// TwinCAT 3 PLC project ExternControl
// ProgramVersion: 3.1.4026.26
// libraries:
//   Tc2_Standard, * (Beckhoff Automation GmbH)
//   Tc2_System, * (Beckhoff Automation GmbH)
//   Tc2_Utilities, * (Beckhoff Automation GmbH)
//   VisuDialogs, * (System)
//   VisuDialogs
// project tree:
//   APPLICATION/ MAIN_APP.TcPOU
//   / GlobalTextList.TcGTLO, MAIN.TcPOU (not stored), PlcTask.TcTTO (not stored), Visualization Manager.TcVMO (not stored)
//   MAPPING/ MAPPING_in.TcPOU (not stored), MAPPING_out.TcPOU (not stored)
//   MAPPING/_types/ U_APP_CTRL.TcDUT (not stored), U_APP_STATE.TcDUT (not stored), U_INSTANCE_CTRL.TcDUT (not stored), U_INSTANCE_STATE.TcDUT (not stored), U_TICKET_LIST_CTRL.TcDUT (not stored), U_TICKET_LIST_DATA_INPUT.TcDUT (not stored), U_TICKET_LIST_DATA_OUTPUT.TcDUT, U_TICKET_LIST_STATE.TcDUT (not stored), U_XTS_STATION_CTRL.TcDUT (not stored), U_XTS_STATION_STATE.TcDUT (not stored), U_XTS_TRANSPORT_CTRL.TcDUT (not stored), U_XTS_TRANSPORT_STATE.TcDUT (not stored)
//   PLC_MOTION/_GVL/ PLC_CONSTANT.TcGVL
//   XTS_TRANSPORT/CaGroup/types/ E_CA_GROUP_STATE.TcDUT, E_GROUP_CHECK.TcDUT, ST_GROUP_INFO.TcDUT
//   XTS_TRANSPORT/ GVL_XTS.TcGVL (not stored), GVL_XTS_CONSTANTS.TcGVL, GVL_XTS_VERSION.TcGVL (not stored)
//   XTS_TRANSPORT/Mover/types/ E_MOVER_CHECK.TcDUT, E_MOVER_CTRL.TcDUT, E_MOVER_SELECTOR.TcDUT, E_MOVER_STATE.TcDUT (not stored), ST_GEAR_DATA.TcDUT, ST_MOVER_CTRL.TcDUT, ST_MOVER_INFO.TcDUT (not stored), ST_MOVER_SELECTOR_CTRL.TcDUT, ST_MOVER_SELECTOR_STATE.TcDUT, ST_MOVER_STATE.TcDUT, ST_MOVE_DATA.TcDUT
//   XTS_TRANSPORT/Xpu/types/ E_XPU_CHECK.TcDUT, E_XPU_CTRL.TcDUT, E_XPU_INIT.TcDUT, E_XPU_STATE.TcDUT, ST_XPU_CTRL.TcDUT, ST_XPU_INFO.TcDUT, ST_XPU_STATE.TcDUT
//   XTS_TRANSPORT/XtsStation/types/ E_STATION_CHECK.TcDUT (not stored), E_STATION_CTRL.TcDUT, E_STATION_GEAR_DISTANCE_AXIS.TcDUT (not stored), E_STATION_STATE.TcDUT (not stored), E_STATION_TYPE.TcDUT (not stored), ST_STATION_CTRL.TcDUT (not stored), ST_STATION_GEAR_PARAMETER.TcDUT (not stored), ST_STATION_LIST_RESULT.TcDUT (not stored), ST_STATION_MOVER_DATA.TcDUT, ST_STATION_PARAMETER.TcDUT, ST_STATION_STATE.TcDUT (not stored), T_NEST_OFFSET.TcDUT (not stored)
//   XTS_TRANSPORT/XtsTransportUnit/types/ E_XTS_TRANSPORT_CHECK.TcDUT, E_XTS_TRANSPORT_CTRL.TcDUT, E_XTS_TRANSPORT_STATE.TcDUT, ST_XTS_TRANSPORT_CTRL.TcDUT, ST_XTS_TRANSPORT_STATE.TcDUT
//   XTS_TRANSPORT/_Visualization/ GROUP_VISU.TcVIS (not stored), MOVER_VISU.TcVIS (not stored), SELECTOR_VISU.TcVIS (not stored), STATION_VISU.TcVIS, XPU_VISU.TcVIS, XTS_TRANSPORT.TcVIS
//   XTS_TRANSPORT/_Visualization/textlists/ TL_E_CTRL_MOVER.TcTLO, TL_E_CTRL_STATION.TcTLO, TL_E_CTRL_TRANSPORT.TcTLO, TL_E_CTRL_XPU.TcTLO
//   XTS_TRANSPORT/_Visualization/types/ ST_XPU_STRINGS.TcDUT (not stored), T_MOVER_SELECTOR.TcVIS
//   _MSG/class/ fb_LocalTime.TcPOU, fb_MessageData.TcPOU, fb_MessageDataCtrl.TcPOU
//   _MSG/ f_MessageSet.TcPOU (not stored), GVL_MSG_AXIS.TcGVL (not stored), GVL_MSG_XTS.TcGVL, I_MessageData.TcIO
//   _MSG/types/ e_Device.TcDUT, E_MessageType.TcDUT, E_MESSAGE_BATCH.TcDUT, E_MESSAGE_CHECK.TcDUT, E_MESSAGE_CTRL.TcDUT (not stored), E_MESSAGE_FLOW.TcDUT, E_MESSAGE_STATE.TcDUT, e_Subdevice.TcDUT, ST_Message.TcDUT, ST_MESSAGE_CTRL.TcDUT (not stored), ST_MESSAGE_STATE.TcDUT (not stored), TL_E_MESSAGETYPE.TcTLO
//   _types/ E_CHECK_STATE.TcDUT, E_PROGRESS.TcDUT, f_GetProgress.TcPOU (not stored), f_GetState.TcPOU
// (motion and I/O tree: see PLC project xtstransport)
// real-time tasks:
//   TASK XTS Task 1: cycle T#250us, priority 1, ADS port 350
//   TASK PLC_1: cycle T#2ms, priority 15, ADS port 353
//   TASK Job Task: cycle default, priority 32
// variable links:
//   ExternControl/ExternControl Instance <-> XtsTransport/XtsTransport Instance
//     PlcTask Inputs/MAIN_APP.eInitXts <-> PlcTask Outputs/MAIN_APP.eInit
//     PlcTask Inputs/MAPPING_in.StationState.byState <-> PlcTask Outputs/MAPPING_XTS_out.StationState.byState
//     PlcTask Inputs/MAPPING_in.TransportState.byState <-> PlcTask Outputs/MAPPING_XTS_out.TransportState.byState
//     PlcTask Outputs/MAPPING_out.StationControl.byCtrl <-> PlcTask Inputs/MAPPING_XTS_in.StationControl.byCtrl
//     PlcTask Outputs/MAPPING_out.TransportControl.byCtrl <-> PlcTask Inputs/MAPPING_XTS_in.TransportControl.byCtrl

// ---- MAPPING/_types/U_TICKET_LIST_DATA_OUTPUT.TcDUT
TYPE U_TICKET_LIST_DATA_OUTPUT :
UNION
  stData              : ST_LIST_NODE_DATA;
  byData   AT %I*     : ARRAY[1..SIZEOF(ST_LIST_NODE_DATA)] OF BYTE;
END_UNION
END_TYPE

// ---- XTS_TRANSPORT/CaGroup/types/E_CA_GROUP_STATE.TcDUT
// {attribute 'qualified_only'}
// {attribute 'strict'}
{attribute 'to_string'}
TYPE E_CA_GROUP_STATE :
(
  // replicated from MC_GROUP_STATE for getting to_string() functionality
	mcGroupStateInvalid   :=0, 
  mcGroupStateDisabled  :=1, 
  mcGroupStateStandby   :=2, 
  mcGroupStateMoving    :=3, 
  mcGroupStateStopping  :=4, 
  mcGroupStateErrorStop :=5, 
  mcGroupStateHoming    :=6, 
  mcGroupStateNotReady  :=7, 
  mcGroupStateSuspended :=8 
)UINT;
END_TYPE

// ---- XTS_TRANSPORT/CaGroup/types/E_GROUP_CHECK.TcDUT
{attribute 'qualified_only'}
{attribute 'to_string'}
TYPE E_GROUP_CHECK :
(
  NULL,
  REFERENCE_GROUP_REF_INVALID := 9000,
  REFERENCE_AXIS_REF_INVALID,
  REFERENCE_CTRL_INVALID,
  REFERENCE_STATE_INVALID,
  REFERENCE_MOVER_ITF_INVALID,
  REFERENCE_XPU_INFO_INVALID,

  CHECK_DONE              := 10000
)UINT;
END_TYPE

// ---- XTS_TRANSPORT/CaGroup/types/ST_GROUP_INFO.TcDUT
TYPE ST_GROUP_INFO :
STRUCT
  GroupStatusValid,
  GroupStatusBusy,
  GroupMoving, 
  GroupHoming, 
  GroupErrorStop, 
  GroupNotReady, 
  GroupStandby, 
  GroupStopping,
 
  GroupDisabled, 
  AllAxesStanding, 
  ConstantVelocity, 
  Accelerating, 
  Decelerating, 
  InPosition, 
  GroupError					  : BIT; 

  GroupErrorId					: UDINT;

  AxisCount      				: UDINT;
  AxisCountEnabled      : UDINT;

  {attribute 'displaymode':='hex'}
  CaGroupOID            : OTCID;

  CaGroupState          : E_CA_GROUP_STATE;
END_STRUCT
END_TYPE

// ---- XTS_TRANSPORT/Mover/types/E_MOVER_CHECK.TcDUT
{attribute 'qualified_only'}
{attribute 'strict'}
{attribute 'to_string'}
TYPE E_MOVER_CHECK :
(
  NULL,
  MOVER_ID_INVALID := 9000,
  REFERENCE_AXIS_REF_INVALID,
  REFERENCE_LAST_POSITION_INVALID,
  REFERENCE_LAST_GAP_INVALID,
  REFERENCE_INFO_INVALID,

  REFERENCE_CTRL_INVALID  := 9100,
  REFERENCE_STATE_INVALID,
  REFERENCE_GEAR_DATA_INVALID,
  REFERENCE_MOVE_DATA_INVALID,
  REFERENCE_MOVER_ITF_INVALID,

  CHECK_DONE  := 10_000
)UINT;
END_TYPE

// ---- XTS_TRANSPORT/Mover/types/E_MOVER_CTRL.TcDUT
{attribute 'qualified_only'}
{attribute 'strict'}
{attribute 'to_string'}
TYPE E_MOVER_CTRL :
(
  MOVER_NULL,               // initial value at startup, used for change of order or retrigger
  MOVER_ENABLE,             // sets MC_Power.Enable
  MOVER_DISABLE,            // removes MC_Power.Enable
  MOVER_MOVE_TO_POS,        // modulo absolute positioning with MC_MoveAbsolute, InTargetPosition check
  MOVER_MOVE_TO_POS_CA,     // modulo absolute positioning with MC_MoveAbsoluteCA, InTargetPosition check
  MOVER_SEND_TO_POS_CA,     // modulo absolute positioning with MC_MoveAbsoluteCA, done after moving ReleaseDistance
  MOVER_HALT,               // halts mover; by use of MC_Halt mover is set passive in CA group
  MOVER_GEAR_IN,            // GearIn for mover in standstill

  MOVER_GEAR_IN_POS_CA,     // GearInPosCA of mover; when FB_GearInPosCa is InSync --> order is done; check SyncDistance yourself and release mover with e_mover_order.mover_SendToPos
  MOVER_GEAR_OUT,           // gear out for mover
  MOVER_RESET,              // MC_RESET for mover
  MOVER_INFO                // used to display MoverInfo in ST_MOVER_SELECTOR_STATE.Info
)UINT;
END_TYPE

// ---- XTS_TRANSPORT/Mover/types/E_MOVER_SELECTOR.TcDUT
{attribute 'qualified_only'}
{attribute 'strict'}
{attribute 'to_string'}
TYPE E_MOVER_SELECTOR :
(
	SELECT_MOVER_INDEX,
  SELECT_MOVER_AXIS_ID
);
END_TYPE

// ---- XTS_TRANSPORT/Mover/types/ST_GEAR_DATA.TcDUT
{attribute 'pack_mode' := '2'}
TYPE ST_GEAR_DATA :
STRUCT
  rDeltaToMasterPos       : LREAL;
  rModuloSyncPosSlave     : LREAL;
  rMasterStartDistance    : LREAL;
  rGearNumerator          : LREAL;
  iGearDenumerator        : USINT  := 1;
END_STRUCT
END_TYPE

// ---- XTS_TRANSPORT/Mover/types/ST_MOVER_CTRL.TcDUT
{attribute 'pack_mode' := '2'}
TYPE ST_MOVER_CTRL :
STRUCT
  Cmd             : E_MOVER_CTRL;  // order to execute on mover
END_STRUCT
END_TYPE

// ---- XTS_TRANSPORT/Mover/types/ST_MOVER_SELECTOR_CTRL.TcDUT
TYPE ST_MOVER_SELECTOR_CTRL :
STRUCT
  Selector      : E_MOVER_SELECTOR; // select by array Index OR AXIS_REF.NcToPlc.AxisId 
  Mover         : UINT;             // array Index OR AXIS_REF.NcToPlc.AxisId
  Control       : ST_MOVER_CTRL;    // mover control struct, put motion command in here

  Data          : ST_MOVE_DATA;     // write your movement parameters
  //Gear          : ST_GEAR_DATA;     // write your gearing parameters
END_STRUCT
END_TYPE

// ---- XTS_TRANSPORT/Mover/types/ST_MOVER_SELECTOR_STATE.TcDUT
TYPE ST_MOVER_SELECTOR_STATE :
STRUCT
  MoverIndex  : UINT;
  AxisId      : UDINT;
  State       : ST_MOVER_STATE;

  Info        : ST_MOVER_INFO;
END_STRUCT
END_TYPE

// ---- XTS_TRANSPORT/Mover/types/ST_MOVER_STATE.TcDUT
{attribute 'pack_mode' := '2'}
TYPE ST_MOVER_STATE :
STRUCT
  State           : E_MOVER_STATE;  // ST_MOVER_CTRL.Cmd with added E_PROGRESS
  MasterId        : USINT;            // mirror NC AxisId of Master axis
END_STRUCT
END_TYPE

// ---- XTS_TRANSPORT/Mover/types/ST_MOVE_DATA.TcDUT
{attribute 'pack_mode' := '2'}
TYPE ST_MOVE_DATA :
STRUCT
  // HAUD 2024 03 14
  // some init data added for example
  rPos            : LREAL :=   2275.0;
  rVelo           : LREAL :=    500.0;
  rAcc            : LREAL :=   5000.0;
  rJerk           : LREAL := 500000.0;
  rGap            : LREAL :=    100.0;
  rOverride       : LREAL :=    100.0;
  rDelta          : LREAL :=      0.05;
  rDistance       : LREAL :=     25.0;
END_STRUCT
END_TYPE

// ---- XTS_TRANSPORT/Xpu/types/E_XPU_CHECK.TcDUT
{attribute 'qualified_only'}
{attribute 'to_string'}
TYPE E_XPU_CHECK :
(
  INIT_CHECK,
  INIT_CHECK_ERROR,
  START_CHECK,
  XPU_INSTANCE_NULL,
  XPU_RAIL_LENGTH,
  GROUP_RAIL_LENGTH,
  RAIL_LENGTH_COMPARE,
  GROUP_NOT_CONFIGURED,
  GROUP_OID_MISMATCH,

  MOVER_COUNT             := 10,
  MOVER_COUNT_ZERO,
  MOVER_COUNT_NOT_EQUAL,

  PROCESSING_UNIT_POSITIONS_VALID         := 20,
  PROCESSING_UNIT_GET_DATA_EXCEED,

  MOVER_ID_STANDARD       := 30,
  MOVER_ID_SIMULATION,
  MOVER_ID_DETECTION_MODE,
  MOVER_ID_DETECTION_VALID,
  MOVER_ID_DETECTION_DC_LINK,
  MOVER_ID_DETECTION_BUSY,
  MOVER_ID_DETECTION_IDLE,
  MOVER_ID_DETECTION_STATE,
  MOVER_ID_MULTIPLE_NOT_SUPPORTED,

  POINTER_CHECK           := 90,
  POINTER_NULL_CTRL,
  POINTER_NULL_STATE,

  CHECK_DONE      := 10_000
)UINT;
END_TYPE

// ---- XTS_TRANSPORT/Xpu/types/E_XPU_CTRL.TcDUT
{attribute 'strict'}
TYPE E_XPU_CTRL :
(
  XTS_CMD_NULL,
  XTS_CMD_INIT                  := 10,
  //XTS_CMD_READ_STN_CONFIG       := 20,
  XTS_IDLE                      := 30
)UINT;
END_TYPE

// ---- XTS_TRANSPORT/Xpu/types/E_XPU_INIT.TcDUT
{attribute 'to_string'}
TYPE E_XPU_INIT :
(
	INIT_START,
  INIT_ENVIRONMENT_OID            := 10,
  INIT_INFO_SERVER_ITF,
  INIT_INFO_SERVER_STATION_COUNT,
  INIT_INFO_SERVER_STATION_OID,
  INIT_CA_GROUP_OID               := 20,
  INIT_CA_GROUP_GET_OID,
  INIT_CA_GROUP_CHECK_OID,
  INIT_CA_GROUP_COM,
  INIT_PARAMETERSET_COUNT,
  INIT_PARAMETERSET_OID,
  INIT_PARAMETERSET_COM,
  INIT_PARAMETERSET_COM_INIT,
  INIT_PARAMETERSET_COM_NEXT,
  INIT_PROCESSING_UNIT_COM        := 30,
  INIT_PROCESSING_UNIT_COM_INIT,
  INIT_PROCESSING_UNIT_PART_COUNT,
  INIT_PROCESSING_UNIT_PART_OID,
  INIT_PROCESSING_UNIT_TRACK_COUNT,
  INIT_PROCESSING_UNIT_TRACK_OID,
  INIT_PROCESSING_UNIT_MOVER_COUNT,
  INIT_PROCESSING_UNIT_MOVER_OID,
  INIT_PROCESSING_UNIT_TASK_COUNT,
  INIT_PROCESSING_UNIT_TASK_OID,
  INIT_TRACK_COM                  := 50,
  INIT_TRACK_COM_INIT,
  INIT_PART_COM                   := 60,
  INIT_PART_COM_INIT,
  INIT_PART_MODULE_COUNT,
  INIT_PART_MODULE_OID,
  INIT_PART_MODULE_COM,
  INIT_PART_MODULE_COM_INIT,
  INIT_PART_MODULE_COM_NEXT,
  INIT_MOVER_COM                  := 70,
  INIT_MOVER_COM_INIT,
  INIT_MOVER_COM_NEXT,
  INIT_NCT_CONTROLLER_OID         := 80,
  INIT_NCT_CONTROLLER_COM,
  INIT_NCT_CONTROLLER_COM_INIT,
  INIT_NCT_BASE_UNIT_COUNT,
  INIT_NCT_BASE_UNIT_ITF,
  INIT_NCT_BASE_UNIT_NEXT,
  INIT_DATA_GET                   := 90,
  INIT_DATA_CHECK,
  INIT_DONE                       := 100
)UINT;
END_TYPE

// ---- XTS_TRANSPORT/Xpu/types/E_XPU_STATE.TcDUT
{attribute 'to_string'}
TYPE E_XPU_STATE :
(
  XTS_NULL,
  XTS_INVALID,
  XTS_INIT                      := 10,    // initialize XPU
  XTS_STATION_INFO_READ         := 20,    // get Station information from Xpu
  XTS_IDLE                      := 30
)UINT;
END_TYPE

// ---- XTS_TRANSPORT/Xpu/types/ST_XPU_CTRL.TcDUT
{attribute 'pack_mode' := '2'}
TYPE ST_XPU_CTRL :
STRUCT
  Cmd             : E_XPU_CTRL;
END_STRUCT
END_TYPE

// ---- XTS_TRANSPORT/Xpu/types/ST_XPU_INFO.TcDUT
{attribute 'pack_mode' := '2'}
TYPE ST_XPU_INFO :
STRUCT
  AllPositionsValid   : BIT;
  IdDetectionError    : BIT;
  IdDetectionValid    : BIT;
  IdDetectionActive   : BIT;

  OperationMode       : UINT;

  IdDetectionMode           : UINT;
  MoverPositionAssignement  : UINT;

  nDetectedAxisCount  : UINT;
  nExpectedAxisCount  : UINT;

  nParameterSetCount  : UINT;
  nModuleCount        : UINT;
  rRailLength         : LREAL;
END_STRUCT
END_TYPE

// ---- XTS_TRANSPORT/Xpu/types/ST_XPU_STATE.TcDUT
{attribute 'pack_mode' := '2'}
TYPE ST_XPU_STATE :
STRUCT
  Init            : E_XPU_INIT;
  State           : E_XPU_STATE;
  Check           : E_XPU_CHECK;  // cyclic check result
  DcLink          : BIT;          // power all motor modules is ON
END_STRUCT
END_TYPE

// ---- XTS_TRANSPORT/XtsStation/types/E_STATION_CTRL.TcDUT
{attribute 'qualified_only'}
{attribute 'strict'}
{attribute 'to_string'}
TYPE E_STATION_CTRL :
(
  STATION_CTRL_NULL,              // nothing happens here
	STATION_INIT            := 1,   // hard reset of station, list is cleared
  STATION_DISABLE         := 10,  // 
  STATION_ENABLE,                 // 

  STATION_MOVER_ENTER     := 20,  // mover may enter station
  STATION_MOVER_ENTER_RETRY,      // retry after E_STATION_STATE.STATION_ERROR_INFEED_ERROR
  STATION_MOVER_SEND,             // do not enter, send to E_STATION_STATE.STATION_MOVER_OUT

  STATION_PROCESS_START   := 30,  // double handshake with extern
  STATION_PROCESS_DONE,           // single handshake with extern
  STATION_PROCESS_NEST_SKIP,

  STATION_MOVER_OUT       := 50,  // mover may leave station now; ticket for mover is checked here (ST_STATION_CTRL.nTargetStation)
  STATION_MOVER_OUT_RETRY,        // retry after E_STATION_STATE.STATION_ERROR_OUTFEED_ERROR

  STATION_MOVER_GONE      := 60   // mover has left station, last handshake station is empty

)USINT;
END_TYPE

// ---- XTS_TRANSPORT/XtsStation/types/ST_STATION_MOVER_DATA.TcDUT
{attribute 'pack_mode' := '2'}
TYPE ST_STATION_MOVER_DATA :
STRUCT
  nMoverId        : USINT;  // who am I?  !! MUST be correct !! - movement to base position sets everything in order, DO NOT manipulate!
  nTargetStation  : USINT;  // where shall I be? used for double checking with StationId at infeed of mover into station

  {attribute 'displaymode':='bin'}
  nMask           : BYTE;   // how many of you are there? (1 = default, no action required)

  rOffset         : REAL;   // offset for use in work flow !! added to static mover offset for every nest(bit) in nMask!!
END_STRUCT
END_TYPE

// ---- XTS_TRANSPORT/XtsStation/types/ST_STATION_PARAMETER.TcDUT
TYPE ST_STATION_PARAMETER :
STRUCT
  eType             : E_STATION_TYPE := 1;  // StationProcess or StationGearInPos
  sText             : STRING(80);           // only description
  rPosWait          : REAL;                 // start of station, 
                                            // a sending station is using this value 
                                            // to send mover to

  rReleaseDistance  : REAL;                 // distance mover has to travel (from ActPos) 
                                            // in order for station to go back to disable

  rGap              : REAL;
  rVelo             : REAL;
  rAccDec           : REAL;
  rJerk             : REAL;

  // how many nests (stop positions) mover has to stop at (1 = default)
  nConfiguredStopCount  : USINT := 1; // 1-8 --> NestMask = BYTE

  // mover stop position in station, relative to rPosWait!!
  rPosStop          : ARRAY[1..8] OF LREAL;
END_STRUCT
END_TYPE

// ---- XTS_TRANSPORT/XtsTransportUnit/types/E_XTS_TRANSPORT_CHECK.TcDUT
{attribute 'qualified_only'}
{attribute 'to_string'}
TYPE E_XTS_TRANSPORT_CHECK :
(
  // info for cyclic checks
  INIT_CHECK,
  START_CHECK,    // check cycle start
  XPU_INIT,       // Xpu: initialization


  // errors in fb_TransportUnit.Check()
  POINTER_CHECK           := 9000,
  POINTER_NULL_CTRL,

  POINTER_NULL_STATE,
  POINTER_NULL_XPU_CTRL,

  POINTER_NULL_XPU_STATE,
  POINTER_NULL_XPU_INFO,

  POINTER_NULL_GROUP_ITF,
  POINTER_NULL_GROUP_INFO,

  POINTER_NULL_MOVER,
  POINTER_NULL_MOVER_ITF,

  POINTER_NULL_MOVER_INFO,
  POINTER_NULL_MOVER_LAST_POS,
  POINTER_NULL_MOVER_LAST_GAP,

  POINTER_NULL_STATION_START,
  POINTER_NULL_STATION_ITF,
  POINTER_NULL_STATION_CONTROL,
  POINTER_NULL_STATION_STATE,
  POINTER_NULL_STATION_CTRL_ITF,

  DONE_CHECK              := 10000
)UINT;
END_TYPE

// ---- XTS_TRANSPORT/XtsTransportUnit/types/E_XTS_TRANSPORT_CTRL.TcDUT
{attribute 'strict'}
{attribute 'to_string'}
TYPE E_XTS_TRANSPORT_CTRL :
(
  CMD_NULL,
  CMD_INIT                  := 10,  // Xpu, Group, Mover initialization: clear errors, clear group, check Xpu data, check mover detection
  CMD_IDLE,

  CMD_MOVER_ENABLE          := 20,  // all mover are enabled, checked for ControlLoopClosed
  CMD_MOVER_DISABLE,                // all mover are disabled, no axis in CaGroup: no error, any axis in CaGroup: group error
  CMD_MOVER_HALT_CA,                // all movers are stopped with MC_HaltCA[]. ONLY use if all movers are in CA group
  CMD_MOVER_STOP,

  CMD_GROUP_CLEAR           := 30,  // halt all movers, clear errors, remove all movers from group, clear group
  CMD_GROUP_BUILD,                  // add all movers to group
  CMD_GROUP_ENABLE,                 // group with movers is enabled
  CMD_GROUP_STOP,                   // moving CA Group is stopped

  CMD_TRANSPORT_START       := 40,  // move all mover[i] to start position
  CMD_TRANSPORT_RESTART             // move all mover[i] to LastPosition[i]

)UINT;
END_TYPE

// ---- XTS_TRANSPORT/XtsTransportUnit/types/E_XTS_TRANSPORT_STATE.TcDUT
{attribute 'to_string'}
TYPE E_XTS_TRANSPORT_STATE :
(
  TRANSPORT_NULL,
  TRANSPORT_INVALID,
  TRANSPORT_INIT            := 10,  // Xpu, Group, Mover initialization: init TcCOM objects, clear errors, clear group, check Xpu data, check mover detection
  TRANSPORT_IDLE,                   // cyclic check for errors, check Xpu data

  TRANSPORT_MOVER_ENABLE    := 20,  // all mover are enabled, checked for ControlLoopClosed
  TRANSPORT_MOVER_DISABLE,          // all mover are disabled
  TRANSPORT_MOVER_HALT_CA,          // all mover standstill
  TRANSPORT_MOVER_STOP,

  TRANSPORT_GROUP_CLEAR     := 30,  // halt all movers, clear errors, remove all movers from group, clear group
  TRANSPORT_GROUP_BUILD,            // add all movers to group
  TRANSPORT_GROUP_ENABLE,           // group with movers is enabled
  TRANSPORT_GROUP_STOP,             // CaGroup Stop, CaGroup Reset, All movers halt

  TRANSPORT_START           := 40,  // move all mover[i] to start position
  TRANSPORT_RESTART                 // move all mover[i] to LastPosition[i]
)UINT;
END_TYPE

// ---- XTS_TRANSPORT/XtsTransportUnit/types/ST_XTS_TRANSPORT_CTRL.TcDUT
{attribute 'pack_mode' := '2'}
TYPE ST_XTS_TRANSPORT_CTRL :
STRUCT
  Cmd       : E_XTS_TRANSPORT_CTRL;
END_STRUCT
END_TYPE

// ---- XTS_TRANSPORT/XtsTransportUnit/types/ST_XTS_TRANSPORT_STATE.TcDUT
{attribute 'pack_mode' := '2'}
TYPE ST_XTS_TRANSPORT_STATE :
STRUCT
  State         : E_XTS_TRANSPORT_STATE;  // combined value of state and result(e_progress); (hint: extract state value by mod division)
  Check         : E_XTS_TRANSPORT_CHECK;

  XpuState      : ST_XPU_STATE;
  XpuInfo       : ST_XPU_INFO;
  GroupInfo     : ST_GROUP_INFO; 
END_STRUCT
END_TYPE

// ---- _MSG/types/e_Device.TcDUT
{attribute 'to_string'}
TYPE e_Device :
(
  Device_Null,                  // NULL               - not to be used
  Device_Main,                  // MAIN(PRG)          - reserved for MAIN(PRG)
  Device_MainAxis,              // MAIN_AXIS(PRG)     - reserved for MAIN_AXIS(PRG)
  Device_Nci,                   // NCI(PRG)           - reserved for NCI(PRG)
  Device_Cam,                   // CAM(PRG            - reserved for CAM(PRG)
  Device_Functions,             // FUNCTIONS(PRG)     - reserved for FUNCTIONS(PRG)
  Device_FlyingSaw,             // FLYING_SAW(PRG)    - reserved for FLYING_SAW(PRG)
  Device_MainApplication,       // MAIN_APP(PRG)      - reserved for MAIN_APP(PRG)

  Device_MoverSelector,         // single mover interface for xts applications
  Device_ParameterSelector,     // fb_ParameterSelector can only exist once in a project.
  Device_Configuration,         // fb_Configuration can handle multiple files therefore only one instance is required
  Device_XmlData,               // generic XML Data (e.g. persistent data)
  Device_Utilities,             // service calls to anyone you may want to talk to, the main intent is to get XPU and TcXtsIo data to the application side

  General           :=  1000,
  CaGroup           :=  2000,
  Xpu               :=  3000,
  XpuCtrl           :=  4000,
  Mover             :=  5000,
  MoverCtrl         :=  6000,
  XtsTransportUnit  :=  7000,
  XfcTriggerBox     :=  8000,
  XfcTouchProbe     :=  9000,
  XtsStation        := 10000,

  Camming           := 11000,
  NciChannel        := 12000,
  NciChannelCtrl    := 13000,
  Axis              := 14000,
  XfcAxis           := 15000,

  // txt file logging LOG_FILE_METRICS
  MetricsXts        := 16000,   //entries from xts Metrics are written into dedicated txt file (see f_MessageSet, here's the diverter)
  MetricsAxis       := 17000,   //entries from PLC_MOTION Metrics are written into dedicated txt file

  // txt file logging LOG_FILE_APP
  Process           := 20000,   // entries from process are written into dedicated txt file.
  ProcessListCtrl   := 21000,
  TicketListCtrl    := 22000,

  Application       := 30000,   // entries from application are written into dedicated txt file.


  // txt file logging LOG_FILE_PRODUCT - this is for you to use
  DataProduct       := 40000
)UDINT;
END_TYPE

// ---- _MSG/types/E_MessageType.TcDUT
{attribute 'strict'}
{attribute 'to_string'}
TYPE E_MessageType :
(
  //-----------------------------------------------------
  //-----------------------------------------------------
  //  message system:
  //  - errors are always calling f_MessageSet()
  //  - errors are always entered into its list
  //
  //  - message severity is set by this enum (like everywhere else)
  //
  //  - message frequency is set by this enum
  //    - IF you get above 50 stations, 
  //      writing to the file system takes time:
  //
  //    Batch: switching on metrics (> Empty) must not add cpu load, 
  //      --> so do not clutter here
  //
  //    Info:  regular flow of information (>Error / >Warning) 
  //           must not add significant cpu load, 
  //      --> so do not clutter here
  //
  //    Verbose and above:
  //    --> for small systems (< 96 mover, < 50 stations) 
  //        you may switch it on for everybody, 
  //        files get big quickly ;-)
  //
  //    --> switch on during test phase for a handful of stations
  //
  //    --> high detail logging always and for everybody
  //    --> we need somebody who transfers data more quickly
  //      --> I can offer a .NET(C#) ADS tool which collects the list.
  //          .NET application then pushes to database
  //-----------------------------------------------------
  //-----------------------------------------------------
  eMessageEmpty,    // he who is without bounds may speak
  eMessageBatch,    // he who counts words, counts numbers (Batch started, Next in Batch, Batch done)
  eMessageError,    // mine, your(')s, anybody's, let the numbers tell you
  eMessageWarning,  // I told you so
  eMessageInfo,     // A long time ago in a galaxy far, far away...
  eMessageVerbose,  // He talks a lot, doesn't he?; Yeah! He's very knowledgeable.
  eMessageSentient  // Keep them out of bright light, Don't get them wet, do not feed them after midnight!! No matter how much they beg!!
)DINT;
END_TYPE

// ---- _MSG/types/E_MESSAGE_BATCH.TcDUT
{attribute 'qualified_only'}
{attribute 'strict'}
{attribute 'to_string'}
TYPE E_MESSAGE_BATCH :
(
	MSG_BATCH_NULL,
  MSG_BATCH_JOB_STARTED,
  MSG_BATCH_NEXT_IN_JOB,
  MSG_BATCH_JOB_DONE
)UINT;
END_TYPE

// ---- _MSG/types/E_MESSAGE_CHECK.TcDUT
{attribute 'qualified_only'}
{attribute 'strict'}
{attribute 'to_string'}
TYPE E_MESSAGE_CHECK :
(
  NULL,
  // 9000 --> here comes your error
  POINTER_INVALID             := 9000,
  POINTER_TIME_INVALID,
  POINTER_LIST_INVALID,
  POINTER_MSG_IDX_INVALID,
  POINTER_ERR_IDX_INVALID,
  POINTER_ROOT_FILE_INVALID,
  POINTER_ROOT_DIR_INVALID,
  POINTER_CTRL_INVALID,
  POINTER_STATE_INVALID,

  // 10000 --> here comes your man
  CHECK_DONE                        := 10000
)UINT;
END_TYPE

// ---- _MSG/types/E_MESSAGE_FLOW.TcDUT
{attribute 'qualified_only'}
{attribute 'strict'}
{attribute 'to_string'}
TYPE E_MESSAGE_FLOW :
(
  MSG_FLOW_INIT,
  MSG_FLOW_ROOT                 := 10,
  MSG_FLOW_ROOT_CREATE,
  MSG_FLOW_ROOT_CREATE_BUSY,
  MSG_FLOW_FOLDER,
  MSG_FLOW_FOLDER_CREATE,
  MSG_FLOW_FOLDER_CREATE_BUSY,
  MSG_FLOW_FILE_CREATE_DONE,
  MSG_FLOW_LINE_START           := 100,
  MSG_FLOW_LINE_BUILD,
  MSG_FLOW_LINE_CHECK,
  MSG_FLOW_WRITE_FILE_BUSY      := 200,
  MSG_FLOW_WRITE_FILE_END,
  MSG_FLOW_WRITE_FILE_DONE      := 1000
)UINT;
END_TYPE

// ---- _MSG/types/E_MESSAGE_STATE.TcDUT
{attribute 'qualified_only'}
//{attribute 'strict'}
{attribute 'to_string'}
TYPE E_MESSAGE_STATE :
(
	MSG_STATE_NULL,
  MSG_STATE_INIT    := 10,
  MSG_STATE_IDLE    := 30,
  MSG_STATE_WRITE   := 50
)UINT;
END_TYPE

// ---- _MSG/types/e_Subdevice.TcDUT
{attribute 'strict'}
{attribute 'to_string'}
TYPE e_Subdevice :
(
  // sub device for message system
  General                 :=  0,
  MainInit,
  // Motion Control FB Instances
  fbPower,
  fbReset,
  fbResetSercos,
  fbHalt,
  fbStop,                 // 5
  fbHome,
  fbJog,
  fbMoveVelocity1,
  fbMoveVelocity2,
  fbMoveAbsolute1,        // 10
  fbMoveAbsolute2,
  fbMoveEndless,
  fbMovePtP,
  fbMoveVelo,
  fbSendToPos,

  // CA CollisionAvoidance FB instances
  // CA group fb instances
  fbCaGroup             := 30,
  fbMoveToPosCa,
  fbSendToAbsPosCa,
  fbSendToModuloPosCa,
  fbGearInPosCa,
  fbGroupAddAxis,
  fbGroupRemoveAxis,
  fbGroupDisable,
  fbGroupEnable,
  fbGroupErrorRead,
  fbGroupStatusRead,
  fbGroupReset,
  fbGroupStop,
  fbHaltCa,

  fbGearIn                := 50,
  fbGearOut,
  fbGearInMultiMaster,

  fbCamOutV2              := 80,
  fbCamInV2,
  fbCamScalingV2,
  fbCamInfoV2,
  fbReadMotionFunction,
  fbReadMotionFunctionPoint,
  fbReadMotionFunctionValues,
  fbWriteMotionFunction,
  fbWriteMotionFunctionPoint,
  fbSetOnlineChangeMode,

  fbReadParameter         := 100,
  fbReadBoolParameter,
  fbWriteParameter,
  fbWriteBoolParameter,
  fbWriteParameterPersistent,
  fbXmlRead,
  fbXmlWrite,
  fbCreateFolder,

  fbBuildGroup            := 200,
  fbClearGroup,
  fbLoadProg,
  fbResetItp,
  fbStartStopItp,
  fbEStopItp,             // 205
  fbStepOnAfterEStopItp,
  fbConfirmHskItp,
  fbDelDtgItp,
  fbNciFeedTablePreparation,
  fbNciFeedTable,         // 210
  fbReadLine,
  fbItpReadRParams,
  fbItpWriteRParams,
  Get_ItpState,
  Get_Error,              // 215


  XfcPositionAtTime       := 300,
  XfcTimeOfPosition,
  XfcTimeToPosition,
  XfcTimeToModuloPosition,
  XfcRecordedPosition,
  XfcTouchProbe,          // 305
  XfcTouchProbeEL1258,
  XfcTouchProbeOptions,
  XfcTriggerRef,
  XfcTriggerRef_MT,
  XfcEl1258Interface_MT,  // 310
  XfcRecordedPosition_MT,
  XfcTriggerOut,
  XfcTriggerStart,
  XfcSwitchOn_2252,
  XfcSwitchOff_2252,      // 315
  XfcInit,
  XfcLatchPosition,
  XfcWaitForPosition,

  AxisMode              := 1000,
  AxisControl,
  AxisStartUp,
  AxisCycle,
  AxisIdle,

  NciControl            := 2000,
  NciStartUp,
  NciCycle,
  NciIdle,

  FlyingSawControl      := 2100,
  FlyingSawStartUp,

  StationLinkedList     := 3000,
  StationInitList,
  StationAddHead,
  StationAddTail,
  StationGetHead,
  StationRemoveHeadValue,
  StationGearInDistanceToSync,
  StationGearInSyncStart,
  StationGearInSyncMove,
  StationGearInSyncEnd,
  StationCalcInfeedPosition,

  StationControl        := 4000,
  StationState, 

  Xpu_fbEnvironment     := 5000,
  Xpu_fbProcessingUnit,
  Xpu_fbXpuPart,
  Xpu_fbXpuTrack,
  Xpu_fbMc2CaGroup,
  Xpu_fbParameterSet,
  Xpu_fbNctController,

  Xpu_fbPartModules     := 5500,

  Xpu_fbMoverXpu        := 6000,

  Xpu_fbNctBaseUnit     := 6500,

  TransportUnit_General := 7000,
  TransportUnit_Restart := 7010,
  TransportUnit_Start,
  TransportUnit_XpuInit,
  TransportUnit_StationClearOutfeed,
  TransportUnit_GroupEnable,
  TransportUnit_GroupClear,
  TransportUnit_GroupBuild,
  TransportUnit_GroupStop,
  TransportUnit_MoverEnableAll,
  TransportUnit_MoverDisableAll,


  CamControl            := 8000,
  CamStartUp,
  CamCycle,

  Process_StationCollector    := 11000,
  Process_ProcessCollector    := 11100,
  Process_ProcessCollector_Init,
  Process_ProcessCollector_Cycle,
  Process_ProcessCollector_Control,

  Process_LinkedList_GetHead,
  Process_LinkedList_RemoveHead,
  Process_LinkedList_AddTail,
  Process_LinkedList_CheckData,
  Process_StationQueue_Check,

  Process_LinkedList_Com              := 11200,
  Process_LinkedList_Com_Init,
  Process_LinkedList_Com_Cmd,
  Process_LinkedList_Com_AddHead,
  Process_LinkedList_Com_AddTail,
  Process_LinkedList_Com_DelHead,
  Process_LinkedList_Com_DelTail,
  Process_LinkedList_Com_GetHead,
  Process_LinkedList_Com_GetTail,


  Instance_Command              := 12000,
  Instance_ProcessConductor,
  Instance_BufferInfeed,
  Instance_Infeed,
  Instance_BufferOutfeed,
  Instance_Outfeed,
  Instance_Sender_Buffer,

  Ticket_LinkedList_Ctrl        := 12100,
  Ticket_LinkedList_Com_Init,
  Ticket_LinkedList_Com_Cmd,
  Ticket_LinkedList_Com_AddHead,
  Ticket_LinkedList_Com_AddTail,
  Ticket_LinkedList_Com_DelHead,
  Ticket_LinkedList_Com_DelTail,
  Ticket_LinkedList_Com_GetHead,
  Ticket_LinkedList_Com_GetTail,
  

  Application                 := 13000,
  Application_Check,
  Application_Clear,
  Application_Cmd,
  Application_Disable,
  Application_Enable,
  Application_Finish,
  Application_Init,
  Application_Proceed,
  Application_Work,

  Utilities                   := 13100,
  Utilities_GetStationOnModule,
  Utilities_SetGlobalConstraints

)DINT;
END_TYPE

// ---- _MSG/types/ST_Message.TcDUT
TYPE ST_Message :
STRUCT
  eType         : e_MessageType;
  eDevice       : e_Device;
  eSubdevice    : e_SubDevice;
  {attribute 'displaymode':='hex'}
  iErrorNumber  : LINT;
  tTime         : STRING(24);
  sText         : STRING(127);
END_STRUCT
END_TYPE

// ---- _types/E_CHECK_STATE.TcDUT
{attribute 'qualified_only'}
{attribute 'strict'}
{attribute 'to_string'}
TYPE E_CHECK_STATE :
(
  CHECK_INIT,
  AXIS_INDEX_OUT_OF_RANGE         :=  10,

	AXIS_REF_POINTER_INVALID        := 100,
  AXIS_CTRL_POINTER_INVALID,
  AXIS_STATE_POINTER_INVALID,
  AXIS_INFO_POINTER_INVALID,
  AXIS_DATA_POINTER_INVALID,
  AXIS_NC_PARAMETER_POINTER_INVALID,
  AXIS_HOME_PARAMETER_POINTER_INVALID,
  AXIS_GEAR_IN_PARAMETER_POINTER_INVALID,
  AXIS_GEAR_IN_MULTIMASTER_POINTER_INVALID,
  AXIS_MOTION_OPTIONS_POINTER_INVALID,

  NCI_NOT_ACTIVATED               := 200,
  NCI_CHANNEL_REF_POINTER_INVALID,
  NCI_AXIS_CONFIG_POINTER_INVALID,
  NCI_MCS_AXIS_POINTER_INVALID,
  NCI_AUX_AXIS_POINTER_INVALID,
  NCI_CTRL_POINTER_INVALID,
  NCI_STATE_POINTER_INVALID,
  NCI_R_PARAMETER_READ_POINTER_INVALID,
  NCI_R_PARAMETER_wRITE_POINTER_INVALID,
  NCI_M_FUNC_POINTER_INVALID,

  CAM_NOT_ACTIVATED               := 300,
  CAM_SLAVE_AXIS_REF_INVALID,
  CAM_SLAVE_ITF_MC_AXIS_INVALID,
  CAM_MASTER_AXIS_REF_INVALID,
  CAM_MOTION_FUNCTION_POINTER_INVALID,
  CAM_MOTION_FUNCTION_POINT_POINTER_INVALID,
  AXIS_LIMIT_SWITCHES_POINTER_INVALID,

  FLYING_SAW_NOT_ACTIVATED        := 400,
  FLYING_SLAVE_ITF_MC_AXIS_INVALID,
  FLYING_MASTER_AXIS_REF_INVALID,
  FLYING_FLY_DATA_POINTER_INVALID,
  FLYING_MOVE_DATA_POINTER_INVALID,
  FLYING_OPTIONS_POINTER_INVALID,
  FLYING_OPTIONS_SYNCMODE_SIZE_NOT_EQUAL,

  PARAMETER_SELECTOR              := 500,
  PARAMETER_SELECTOR_CTRL_REF_INVALID,
  PARAMETER_SELECTOR_STATE_REF_INVALID,
  PARAMETER_SELECTOR_AXIS_ITF_INVALID,


  CHECK_DONE                      := 10000
  
)UINT;
END_TYPE

// ---- _types/E_PROGRESS.TcDUT
{attribute 'qualified_only'}
//{attribute 'strict'}
{attribute 'to_string'}
TYPE E_PROGRESS :
(
  // progress has 2 use cases
  // 1. as offset to cyclic interface's state 
  //    for the requested command/function
  //    e.g. State := <Enum equivalent to eCmd> + E_PROGRESS
  //
  // 2. as state feedback (result) from (any) method
  PROGRESS_INVALID,
  PROGRESS_NOT_EXIST      :=   100,
  PROGRESS_INIT           :=  1000,
  PROGRESS_BUSY           :=  2000,
  PROGRESS_PREPARE        :=  3000,
  PROGRESS_STARTUP        :=  4000,
  PROGRESS_CHECK          :=  5000,
  PROGRESS_OCCUPIED       :=  6000,
  PROGRESS_WORKING        :=  7000,
  PROGRESS_STILL_WORKING  :=  8000,
  PROGRESS_ERROR          :=  9000,
  PROGRESS_DONE           := 10000
)UINT;
END_TYPE

// ---- PLC_MOTION/_GVL/PLC_CONSTANT.TcGVL
//{attribute 'qualified_only'}
VAR_GLOBAL CONSTANT


  //-----------------------------------------------------------------------------
  // AXIS related limits
  //-----------------------------------------------------------------------------
  MAX_AXIS              : UINT    := 3;
  MAX_RETRY             : UINT    := 5;


  //-----------------------------------------------------------------------------
  // NCI related limits and *.nc standard folder
  //-----------------------------------------------------------------------------
{IF NOT defined (BSD)}
  NCI_DIR               : STRING  := 'C:\TwinCAT\Mc\Nci\';
{ELSE}
  NCI_DIR               : STRING  := '/usr/local/etc/TwinCAT/Mc/Nci/';
{END_IF}

{IF defined (NCI)}
  {info 'PLC_MOTION_LAYER: NCI'}
  NCI_ACTIVE            : BOOL    := TRUE;
  CONFIG_NAME           : STRING  := 'NCI_Spec_Ch_';
{ELSE}
  NCI_ACTIVE            : BOOL    := FALSE;
  CONFIG_NAME           : STRING  := 'NCI_NOT_ACTIVE';
{END_IF}

  MAX_NCI_CH            : UINT    := 1;

  MAX_PATH_STEPS        : UINT    := 5;
  MAX_MC_AXIS           : UINT    := 3;
  MAX_AUX_AXIS          : UINT    := 2;
  MAX_R_PARA            : UINT    := 10;


  //-----------------------------------------------------------------------------
  // CAMMING related limits
  //-----------------------------------------------------------------------------
{IF defined (CAM)}
  {info 'PLC_MOTION_LAYER: CAM'}
  CAM_ACTIVE                  : BOOL    := TRUE;
{ELSE}
  CAM_ACTIVE                  : BOOL    := FALSE;
{END_IF}

  MAX_CAM_CH                  : UINT    := 1;

  MAX_MOTION_FUNCTION_POINTS  : UINT    := 10;

  // HAUD
  // 17.07.2024
  // Start Implementation of Position Trigger function
  //  - Timestamp/position output
  //  - Latch DC time from input
  
  MAX_TRIGGER_BOX             : UINT := 12;
  MAX_TOUCH_PROBE             : UINT := 12;
  MAX_TRIGGER_COUNT           : UINT :=  4;
  MAX_MTI_CH                  : UINT :=  1; // MAX mti channel per EL terminal

{IF defined (XFC)}
  {info 'PLC_MOTION_LAYER: XFC'}
  XFC_ACTIVE                  : BOOL := TRUE;
{ELSE}
  XFC_ACTIVE                  : BOOL := FALSE;
{END_IF}

  // HAUD
  // 2026 05 28
  // Gear In Pos implementation for flying saw application 

{IF defined (SAW)}
  {info 'PLC_MOTION_LAYER: FLYING_SAW'}
  FLY_SAW_ACTIVE              : BOOL  := TRUE;
{ELSE}
  FLY_SAW_ACTIVE              : BOOL  := FALSE;
{END_IF}
END_VAR

// ---- XTS_TRANSPORT/GVL_XTS_CONSTANTS.TcGVL
//{attribute 'qualified_only'}
VAR_GLOBAL CONSTANT
//-----------------------------------------------------------------------------------------------------------------------------------------
//-----------------------------------------------------------------------------------------------------------------------------------------
//
//  HAUD 2026.03.15
//  - parameter list deleted (never used the parameter feature anyway), 
//    back to static global constants
//
//-----------------------------------------------------------------------------------------------------------------------------------------
//-----------------------------------------------------------------------------------------------------------------------------------------
//  Connections to XTS Utility Lib data: 
//  - suits this simple approach, 
//  - leaves you options to expand, 
//  - expansion and multiplication is not implemented here on purpose, 
//  - this project is designed to get the main ideas across, 
//  - setting up a matrix for multiple fb_Xpu instances with it, 
//    --> a second step you might want to organize from here; 
//        --> I leave the details up to you
//-----------------------------------------------------------------------------------------------------------------------------------------
//-----------------------------------------------------------------------------------------------------------------------------------------
  MAX_MOVER             : UINT    := 10;
//   MAX_MOVER           : UINT    := TO_UINT(Tc3_XTS_Utility.TcIoXtsEnvironmentParameterList.MaxXtsMoversPerXpu);
//   MAX_MODULE          : UINT    := TO_UINT(Tc3_XTS_Utility.TcIoXtsEnvironmentParameterList.MaxModulesPerPart);
//   MAX_PART            : UINT    := TO_UINT(Tc3_XTS_Utility.TcIoXtsEnvironmentParameterList.MaxXtsPartsPerXpu);
//   MAX_TRACK           : UINT    := TO_UINT(Tc3_XTS_Utility.TcIoXtsEnvironmentParameterList.MaxXtsTracksPerXpu);
//   MAX_GROUP           : UINT    := TO_UINT(Tc3_XTS_Utility.TcIoXtsEnvironmentParameterList.MaxXtsCaGroup);
// 
//   MAX_INFO_SERVER     : UINT    := TO_UINT(Tc3_XTS_Utility.TcIoXtsEnvironmentParameterList.MaxXtsInfoServer);
//   MAX_INFO_STATION    : UINT    := TO_UINT(Tc3_XTS_Utility.TcIoXtsEnvironmentParameterList.MaxXtsInfoStation);
//   MAX_INFO_STOP_POS   : UINT    := TO_UINT(Tc3_XTS_Utility.TcIoXtsEnvironmentParameterList.MaxXtsStopPositionsPerStation);
// 
//   MAX_PARAMETER_SET   : UINT    := TO_UINT(Tc3_XTS_Utility.TcIoXtsEnvironmentParameterList.MaxXtsParameterSet);
// 
//   MAX_NCT_BASE_UNIT   : UINT    := TO_UINT(Tc3_XTS_Utility.TcIoXtsEnvironmentParameterList.MaxXtsNctBaseUnitInterfaces);
//-----------------------------------------------------------------------------------------------------------------------------------------
//-----------------------------------------------------------------------------------------------------------------------------------------
//  XTS_TRANSPORT_LAYER
//  - project constants you will have to adjust in order to build your transport logic
//-----------------------------------------------------------------------------------------------------------------------------------------
//-----------------------------------------------------------------------------------------------------------------------------------------
  MAX_STATION         : UINT    := 5;

  MAX_STATION_NEST    : UINT    := TO_UINT(SIZEOF(ST_STATION_STATE.nMask)*8);
  MAX_LIST_NODES      : UINT    := MAX_MOVER;
  MAX_MASTER          : UINT    := 1;
//-----------------------------------------------------------------------------------------------------------------------------------------
//-----------------------------------------------------------------------------------------------------------------------------------------
END_VAR

// ---- _MSG/GVL_MSG_XTS.TcGVL
{attribute 'qualified_only'}
VAR_GLOBAL CONSTANT
  //-----------------------------------------------------------------------------
  // file paths for message system
  //  - compiler define option WIN switches to Windows file paths
  //-----------------------------------------------------------------------------
{IF defined (WIN)}
  {info 'WIN folders'}
  LOG_DIR               : STRING  := 'C:\TwinCAT\#MsgFiles\';       // delimiter at the end is mandatory!!
  CON_DIR               : STRING  := 'C:\TwinCAT\#Configuration\';  // delimiter at the end is mandatory!!
{ELSE}
  {info 'BSD folders'}
  LOG_DIR               : STRING  := '/usr/local/etc/TwinCAT/#MsgFiles/';       // delimiter at the end is mandatory!!
  CON_DIR               : STRING  := '/usr/local/etc/TwinCAT/#Configuration/';  // delimiter at the end is mandatory!!
{END_IF}

  LOG_FILE              : STRING  := 'MSG_XtsTransport_';
  LOG_FILE_APP          : STRING  := 'MSG_Application_';
  LOG_FILE_METRIC       : STRING  := 'MSG_XtsTransportMetrics_';

  MAX_MESSAGE           : UINT    := 2000; // max entry in message list
END_VAR
VAR_GLOBAL
  //-----------------------------------------------------------------------------
  // Message System
  //  - Everybody uses f_MessageSet(ST_Message)
  //    - DECISION WHICH LIST IS MADE IN f_MessageSet !!
  //    - which list to use is determined by e_Device in your message
  //
  //  - MessageData instances are self sufficient and need only 
  //    datafield assignment for correct data-flow
  //
  //
  //-----------------------------------------------------------------------------
  //-----------------------------------------------------------------------------
  //-----------------------------------------------------------------------------
  // (ST_Message.eDevice := e_Device.Application)
  //----------------------------------------------------------------------------- 
  ApplicationMessageData          : fb_MessageDataCtrl;
  ApplicationMessageCtrl          : st_message_ctrl;
  ApplicationMessageState         : st_message_state;

  ApplicationMessages             : ARRAY[1..MAX_MESSAGE] OF ST_Message;
  MessageApplicationIndex         : UINT := 0; // message index for higher layers (grouping, Instances, etc.)
  MessageApplicationError         : UINT := 0; // error counter for higher learning
  //-----------------------------------------------------------------------------
  //-----------------------------------------------------------------------------
  // (ST_Message.eDevice := from Device_Null to XfcAxis)
  //-----------------------------------------------------------------------------
  TransportMessageData            : fb_MessageDataCtrl;
  TransportMessageCtrl            : st_message_ctrl;
  TransportMessageState           : st_message_state;

  TransportMessages               : ARRAY[1..MAX_MESSAGE] OF ST_Message;
  MessageTransportIndex           : UINT := 0; // message index for base layer
  MessageTransportError           : UINT := 0; // error counter for base layer
  //-----------------------------------------------------------------------------
  //-----------------------------------------------------------------------------
  // (ST_Message.eDevice := e_Device.Metrics)
  //-----------------------------------------------------------------------------
  MetricsMessageData              : fb_MessageDataCtrl;
  MetricsMessageCtrl              : st_message_ctrl;
  MetricsMessageState             : st_message_state;

  MetricsMessages                 : ARRAY[1..MAX_MESSAGE] OF ST_Message;
  MessageMetricsIndex             : UINT := 0; // message index for metrics data
  MessageMetricsError             : UINT := 0; // error counter for metrics data
  //-----------------------------------------------------------------------------
  //-----------------------------------------------------------------------------
  // (ST_Message.eDevice := e_Device.ProductData)
  //-----------------------------------------------------------------------------
  ProductMessageData              : fb_MessageDataCtrl;   // This is for you
  ProductMessageCtrl              : st_message_ctrl;
  ProductMessageState             : st_message_state;

  ProductMessages                 : ARRAY[1..MAX_MESSAGE] OF ST_Message;
  MessageProductIndex             : UINT := 0; // message index for your product data
  MessageProductError             : UINT := 0; // error counter for your product data
  //-----------------------------------------------------------------------------
  //-----------------------------------------------------------------------------
  fbLocalTime                     : fb_LocalTime;
  dtLocalTime                     : DT;
  sLocalTime                      : STRING;
  //-----------------------------------------------------------------------------
  //-----------------------------------------------------------------------------
  //-----------------------------------------------------------------------------
  //-----------------------------------------------------------------------------
  MessageLevelXpu                 : E_MessageType;
  MessageLevelStations            : ARRAY[1..MAX_STATION] OF E_MessageType;
  MessageLevelMovers              : ARRAY[1..MAX_MOVER]   OF E_MessageType;

  //MessageLevelProcess             : ARRAY[1..MAX_PROCESS] OF E_MessageType;

{IF defined (TEST)}
  {info 'TEST logging enabled'}
  MessageLevel                    : E_MessageType := eMessageinfo; // a lot of messages
{ELSE}
  MessageLevel                    : E_MessageType := eMessageEmpty; // only errors are written into list 
{END_IF}

END_VAR

// ---- _MSG/I_MessageData.TcIO
INTERFACE I_MessageData

PROPERTY DirRoot : POINTER to string(255)
SET
END_SET
END_PROPERTY

PROPERTY ErrorIndex : reference to uint
SET
END_SET
END_PROPERTY

PROPERTY FileRoot : pointer to string(255)
SET
END_SET
END_PROPERTY

PROPERTY LocalTime : pointer to DT
SET
END_SET
END_PROPERTY

PROPERTY MessageIndex : reference to uint
SET
END_SET
END_PROPERTY

PROPERTY MsgList : pointer to ARRAY[1..GVL_MSG_XTS.MAX_MESSAGE] OF st_message
SET
END_SET
END_PROPERTY

END_INTERFACE

// ---- _MSG/class/fb_MessageDataCtrl.TcPOU
FUNCTION_BLOCK fb_MessageDataCtrl EXTENDS fb_MessageData
VAR
  _stCtrl       : REFERENCE TO ST_MESSAGE_CTRL;
  _stState      : REFERENCE TO ST_MESSAGE_STATE;

  _eCmd,
  _eCmdOld      : E_MESSAGE_CTRL;

  _eResult,
  _eJobResult   : E_PROGRESS;

  _eState       : E_MESSAGE_STATE;

END_VAR

//-----------------------------------------------------------------------------
// check pointers
//-----------------------------------------------------------------------------
IF NOT Check()
THEN
  _eResult                      := E_PROGRESS.PROGRESS_ERROR;
  RETURN;
END_IF
//-----------------------------------------------------------------------------
// check date
// new message file for a new day
//-----------------------------------------------------------------------------
IF (FolderDate(_dtLocalTime) <> _sFolderDate)
THEN
  _bFileCreated                 := FALSE;
END_IF
//-----------------------------------------------------------------------------
//----------------------------------------------------------------------------- 
// copy to local for debug
_eCmd                         := _stCtrl.Cmd;

// cyclic check for command change
// get state for cmd
IF (_eCmd <> _eCmdOld)
THEN
  // get matching sdtate for Ctrl.Cmd
  _eState                     := Cmd(_eCmd);
  _eCmdOld                    := _eCmd;
END_IF


CASE _eResult
OF
  E_PROGRESS.PROGRESS_INVALID:
    _stState.State            := E_MESSAGE_STATE.MSG_STATE_NULL;

  E_PROGRESS.PROGRESS_ERROR:
    _stState.State            := _eState + E_PROGRESS.PROGRESS_ERROR;

  E_PROGRESS.PROGRESS_DONE:
    _stState.State            := _eState + E_PROGRESS.PROGRESS_DONE;

ELSE
  // work in progress
  // update progress for extern use
  _stState.State              := _eState + _eResult;

  CASE _eState
  OF
    E_MESSAGE_STATE.MSG_STATE_INIT:
      _eResult                := BuildFolder(TRUE);


    E_MESSAGE_STATE.MSG_STATE_IDLE:
      IF (_nMsgIndex < GVL_MSG_XTS.MAX_MESSAGE - GVL_MSG_XTS.MAX_MESSAGE/10)
      THEN
        _eResult              := E_PROGRESS.PROGRESS_WORKING;
      ELSE
        _eResult              := E_PROGRESS.PROGRESS_DONE;
        _nMsgIndex            := 0;
        // copy from attached list to local
        memcpy(ADR(_aWriteList), _pMsgList, SIZEOF(_aWriteList));
        // clear attached list
        memset(_pMsgList, 0, SIZEOF(_aWriteList));
      END_IF


    E_MESSAGE_STATE.MSG_STATE_WRITE:
      _eResult                := BuildFileData(TRUE);

  ELSE
      _eResult               := E_PROGRESS.PROGRESS_INVALID;
  END_CASE
END_CASE

METHOD BuildFileData : e_progress
VAR_INPUT
  Execute     : BOOL;
END_VAR
VAR_INST
  _nErrorId   : UDINT;
  _eState,
  _eRes       : E_PROGRESS;
  _eFlow      : E_MESSAGE_FLOW;

  _nStringLength  : UINT;
END_VAR
//-----------------------------------------------------------------------------
IF NOT Execute 
THEN
  _eRes                           := WriteData(FALSE);
  _eRes                           := BuildFolder(FALSE);
	_eState                         := E_PROGRESS.PROGRESS_INIT; 
END_IF 
//-----------------------------------------------------------------------------
IF NOT Check() 
THEN 
	BuildFileData                   := E_PROGRESS.PROGRESS_ERROR; 
	RETURN; 
END_IF
//-----------------------------------------------------------------------------
//-----------------------------------------------------------------------------
CASE _eState
OF
  E_PROGRESS.PROGRESS_INIT:
    IF Execute
    THEN
      _nErrorId                   := 0;
      _iStart 	                  := 1;
      _iEnd 		                  := SEL((_nMsgIndex > GVL_MSG_XTS.MAX_MESSAGE-1),
                                          _nMsgIndex,
                                          GVL_MSG_XTS.MAX_MESSAGE);

      memset(ADR(_sWriteData),0,SIZEOF(_sWriteData));

      IF (_sFolderDate <> FolderDate(_dtLocalTime))
      THEN
        _eState                   := E_PROGRESS.PROGRESS_PREPARE;
      ELSE
        _eState                   := E_PROGRESS.PROGRESS_BUSY;
        _eFlow                    := E_MESSAGE_FLOW.MSG_FLOW_LINE_START;
      END_IF
    END_IF
END_CASE
//-----------------------------------------------------------------------------
//-----------------------------------------------------------------------------
CASE _eState
OF
  E_PROGRESS.PROGRESS_PREPARE:
    _eRes                         := BuildFolder(TRUE);
    CASE _eRes
    OF
      E_PROGRESS.PROGRESS_DONE:
      _eState                     := E_PROGRESS.PROGRESS_BUSY;
      _eFlow                      := E_MESSAGE_FLOW.MSG_FLOW_LINE_START;

      E_PROGRESS.PROGRESS_ERROR:
      _eState                     := E_PROGRESS.PROGRESS_ERROR;
    END_CASE
END_CASE
//-----------------------------------------------------------------------------
//-----------------------------------------------------------------------------
CASE _eState
OF
  E_PROGRESS.PROGRESS_BUSY:
  CASE _eFlow
  OF
    E_MESSAGE_FLOW.MSG_FLOW_LINE_START:
      _eRes                       := BuildFolder(FALSE);
      _nErrIndex                  := 0; // rise and shine, all quarrels erased but not forgotten
      _nMsgIndex                  := 0;
  
      // copy from attached list to local
      memcpy(ADR(_aWriteList), _pMsgList, SIZEOF(_aWriteList));
  
      // clear attached list
      memset(_pMsgList, 0, SIZEOF(_aWriteList));


      _eFlow                      := E_MESSAGE_FLOW.MSG_FLOW_LINE_BUILD;
      _iCount                     := _iStart;
  END_CASE
  CASE _eFlow
  OF
    E_MESSAGE_FLOW.MSG_FLOW_LINE_BUILD:
      _eFlow                      := E_MESSAGE_FLOW.MSG_FLOW_LINE_CHECK;
      IF (_aWriteList[_iCount].eType > E_MessageType.eMessageEmpty)
      THEN
        _sTmp                     := TO_STRING(_aWriteList[_iCount].eType);
        _sTmp                     := Tc2_Standard.CONCAT(_sTmp, _sTab);
        _sTmp                     := Tc2_Standard.CONCAT(_sTmp, _aWriteList[_iCount].tTime);
        _sTmp                     := Tc2_Standard.CONCAT(_sTmp, _sTab);
        _sTmp                     := Tc2_Standard.CONCAT(_sTmp, Device_To_String(_aWriteList[_iCount].eDevice));
        _sTmp                     := Tc2_Standard.CONCAT(_sTmp, _sTab);
        _sTmp                     := Tc2_Standard.CONCAT(_sTmp, TO_STRING(_aWriteList[_iCount].eSubdevice));
        _sTmp                     := Tc2_Standard.CONCAT(_sTmp, _sTab);
        _sTmp                     := Tc2_Standard.CONCAT(_sTmp, TO_STRING(_aWriteList[_iCount].iErrorNumber));
        _sTmp                     := Tc2_Standard.CONCAT(_sTmp, _sTab);
        _sTmp                     := Tc2_Standard.CONCAT(_sTmp, _aWriteList[_iCount].sText);
        _sTmp                     := Tc2_Standard.CONCAT(_sTmp, _sNewLine);
        Builder(ADR(_sTmp), ADR(_sWriteData), StringLen(ADR(_sTmp)));
      END_IF
      _iCount                     := _iCount + 1;
  END_CASE
  CASE _eFlow
  OF
    E_MESSAGE_FLOW.MSG_FLOW_LINE_CHECK:
    IF NOT (_iCount > _iEnd)
    THEN
      _eFlow                      := E_MESSAGE_FLOW.MSG_FLOW_LINE_BUILD;
    ELSE
      _eState                     := E_PROGRESS.PROGRESS_WORKING;
      _eFlow                      := E_MESSAGE_FLOW.MSG_FLOW_WRITE_FILE_BUSY;
    END_IF
  END_CASE
END_CASE
//-----------------------------------------------------------------------------
//-----------------------------------------------------------------------------
CASE _eState
OF
  E_PROGRESS.PROGRESS_WORKING:
  CASE _eFlow
  OF
    E_MESSAGE_FLOW.MSG_FLOW_WRITE_FILE_BUSY:
      _nStringLength              := StringLen(ADR(_sWriteData));
      IF NOT (_nStringLength > 1)
      THEN
        _eState                   := E_PROGRESS.PROGRESS_DONE; 
       _eFlow                     := E_MESSAGE_FLOW.MSG_FLOW_WRITE_FILE_DONE;
      ELSE
        _eFlow                    := E_MESSAGE_FLOW.MSG_FLOW_WRITE_FILE_END;
        _eRes                     := WriteData(FALSE);
      END_IF
  END_CASE
  CASE _eFlow
  OF
    E_MESSAGE_FLOW.MSG_FLOW_WRITE_FILE_END:
      _eRes                       := WriteData(TRUE);

      IF (_eRes = E_PROGRESS.PROGRESS_ERROR)
      THEN
        _eState                   := E_PROGRESS.PROGRESS_ERROR;

      ELSIF (_eRes = E_PROGRESS.PROGRESS_DONE)
      THEN
        _eState                   := E_PROGRESS.PROGRESS_DONE;
        _eFlow                    := E_MESSAGE_FLOW.MSG_FLOW_WRITE_FILE_DONE;
        _eRes                     := WriteData(FALSE);
      END_IF
  END_CASE
END_CASE
//-----------------------------------------------------------------------------
//-----------------------------------------------------------------------------

BuildFileData                     := _eState;
END_METHOD

METHOD BuildFolder : e_progress
VAR_INPUT
  Execute           : BOOL;
END_VAR
VAR_INST
  _nErrorId   : UDINT;
  _eState     : E_PROGRESS;
  _eFlow      : E_MESSAGE_FLOW;
END_VAR
//-----------------------------------------------------------------------------
IF NOT Execute 
THEN 
	_eState                       := E_PROGRESS.PROGRESS_INIT; 
END_IF 
//-----------------------------------------------------------------------------
IF NOT Check() 
THEN 
	BuildFolder                   := E_PROGRESS.PROGRESS_ERROR; 
	RETURN; 
END_IF
//-----------------------------------------------------------------------------
//-----------------------------------------------------------------------------
CASE _eState
OF
  E_PROGRESS.PROGRESS_INIT:
    IF Execute
    THEN
      _nErrorId                 := 0;
      _bFileCreated             := FALSE;

      _sFolderDate              := FolderDate(_dtLocalTime);
      _eState                   := E_PROGRESS.PROGRESS_BUSY;
      _eFlow                    := E_MESSAGE_FLOW.MSG_FLOW_ROOT;
    END_IF
END_CASE
//-----------------------------------------------------------------------------
//-----------------------------------------------------------------------------
CASE _eState
OF
  E_PROGRESS.PROGRESS_BUSY:
  CASE _eFlow
  OF
    E_MESSAGE_FLOW.MSG_FLOW_ROOT:
      _eFlow                    := E_MESSAGE_FLOW.MSG_FLOW_ROOT_CREATE;
      _fbCreateDir.sPathName    := left(_pDirRoot^,len(_pDirRoot^)-1);
      _fbCreateDir(
              bExecute	        := FALSE);
    
    E_MESSAGE_FLOW.MSG_FLOW_ROOT_CREATE:
      (* create root folder *)
      _fbCreateDir(
              bExecute	        := TRUE);
      IF _fbCreateDir.bBusy
      THEN
        _eFlow                  := E_MESSAGE_FLOW.MSG_FLOW_ROOT_CREATE_BUSY;
      END_IF
    
    E_MESSAGE_FLOW.MSG_FLOW_ROOT_CREATE_BUSY:
      _fbCreateDir(
              bExecute	        := TRUE);
      IF NOT _fbCreateDir.bBusy
      THEN
        _eState                 := E_PROGRESS.PROGRESS_PREPARE;
        _eFlow                  := E_MESSAGE_FLOW.MSG_FLOW_FOLDER;
      END_IF
  END_CASE
END_CASE
//-----------------------------------------------------------------------------
//-----------------------------------------------------------------------------
CASE _eState
OF
  E_PROGRESS.PROGRESS_PREPARE:
  CASE _eFlow
  OF
    E_MESSAGE_FLOW.MSG_FLOW_FOLDER:
      _eFlow                    := E_MESSAGE_FLOW.MSG_FLOW_FOLDER_CREATE;
      _sFolderDate              := FolderDate(_dtLocalTime);
      _fbCreateDir.sPathName    := concat(_pDirRoot^, _sFolderDate);
      _fbCreateDir(
              bExecute	        := FALSE);
  
    E_MESSAGE_FLOW.MSG_FLOW_FOLDER_CREATE:
      (* create active folder *)
      _fbCreateDir(
              bExecute	        := TRUE);
      IF _fbCreateDir.bBusy
      THEN
        _eFlow                  := E_MESSAGE_FLOW.MSG_FLOW_FOLDER_CREATE_BUSY;
      END_IF
    
    E_MESSAGE_FLOW.MSG_FLOW_FOLDER_CREATE_BUSY:
      _fbCreateDir(
              bExecute	        := TRUE);
      IF NOT _fbCreateDir.bBusy
      THEN
        _eState                 := E_PROGRESS.PROGRESS_CHECK;
        _eFlow                  := E_MESSAGE_FLOW.MSG_FLOW_FILE_CREATE_DONE;
        _fbCreateDir(
                bExecute	      := FALSE);
      END_IF
  END_CASE
END_CASE
//-----------------------------------------------------------------------------
//-----------------------------------------------------------------------------
CASE _eState
OF
  E_PROGRESS.PROGRESS_CHECK:
  CASE _eFlow
  OF
    E_MESSAGE_FLOW.MSG_FLOW_FILE_CREATE_DONE:
      _eState                   := E_PROGRESS.PROGRESS_DONE;
      _bFileCreated             := TRUE;

      // build complete file path
      _sTmp                     := concat(concat(_pFileRoot^, _sFolderDate),'.txt');
      _sTmp                     := concat('\', _sTmp);
      _sFilename                := concat(_fbCreateDir.sPathName, _sTmp);
  END_CASE
END_CASE

BuildFolder                     := _eState;
END_METHOD

METHOD Check : BOOL
VAR_INPUT
END_VAR

IF NOT __ISVALIDREF(_stCtrl)
THEN
  _eCheck       := E_MESSAGE_CHECK.POINTER_CTRL_INVALID;
  RETURN;
END_IF

IF NOT __ISVALIDREF(_stState)
THEN
  _eCheck       := E_MESSAGE_CHECK.POINTER_STATE_INVALID;
  RETURN;
END_IF
//-----------------------------------------------------------------
//-----------------------------------------------------------------
IF NOT (_dtLocalTime <> 0)
THEN
  _eCheck       := E_MESSAGE_CHECK.POINTER_TIME_INVALID;
  RETURN;
END_IF

IF NOT (_pMsgList <> 0)
THEN
  _eCheck       := E_MESSAGE_CHECK.POINTER_LIST_INVALID;
  RETURN;
END_IF

IF NOT (_pFileRoot <> 0)
THEN
  _eCheck       := E_MESSAGE_CHECK.POINTER_ROOT_FILE_INVALID;
  RETURN;
END_IF

IF NOT (_pDirRoot <> 0)
THEN
  _eCheck       := E_MESSAGE_CHECK.POINTER_ROOT_DIR_INVALID;
  RETURN;
END_IF

IF NOT __ISVALIDREF(_nMsgIndex)
THEN
  _eCheck       := E_MESSAGE_CHECK.POINTER_MSG_IDX_INVALID;
  RETURN;
END_IF

IF NOT __ISVALIDREF(_nErrIndex)
THEN
  _eCheck       := E_MESSAGE_CHECK.POINTER_ERR_IDX_INVALID;
  RETURN;
END_IF


_eCheck         := E_MESSAGE_CHECK.CHECK_DONE;
Check           := TRUE;
END_METHOD

METHOD Cmd : e_message_state
VAR_INPUT
  Command     : e_message_ctrl;
END_VAR


CASE Command
OF
  E_MESSAGE_CTRL.MSG_CTRL_NULL:
    _eResult                    := E_PROGRESS.PROGRESS_INVALID;
    Cmd                         := E_MESSAGE_STATE.MSG_STATE_NULL;

  E_MESSAGE_CTRL.MSG_CTRL_INIT:
    _eResult                    := BuildFolder(FALSE);
    Cmd                         := E_MESSAGE_STATE.MSG_STATE_INIT;

  E_MESSAGE_CTRL.MSG_CTRL_IDLE:
    _eResult                    := BuildFileData(FALSE);
    Cmd                         := E_MESSAGE_STATE.MSG_STATE_IDLE;

  E_MESSAGE_CTRL.MSG_CTRL_WRITE:
    _eResult                    := BuildFileData(FALSE);
    Cmd                         := E_MESSAGE_STATE.MSG_STATE_WRITE;
    IF (_nMsgIndex = 0)
    THEN
       // go back to sleep
      _eResult                := E_PROGRESS.PROGRESS_DONE;
    END_IF
ELSE
    //_eResult                    := E_PROGRESS.PROGRESS_ERROR;
    Cmd                         := E_MESSAGE_STATE.MSG_STATE_NULL;
END_CASE
END_METHOD

PROPERTY Ctrl : REFERENCE to ST_MESSAGE_CTRL
SET
_stCtrl ref= Ctrl;
END_SET
END_PROPERTY

PROPERTY FileCreated : bool
GET
FileCreated := _bFileCreated;
END_GET
END_PROPERTY

PROPERTY State : REFERENCE TO ST_MESSAGE_STATE
SET
_stState ref= State;
END_SET
END_PROPERTY

END_FUNCTION_BLOCK

// ---- _MSG/class/fb_MessageData.TcPOU
FUNCTION_BLOCK ABSTRACT fb_MessageData IMPLEMENTS I_MessageData
VAR CONSTANT
{attribute 'hide'}
  STR_LEN       : UDINT := 524_288;
END_VAR
VAR
  _eCheck       : E_MESSAGE_CHECK;            // pointer check state

  _pFileRoot    : POINTER TO STRING(255);     // you decide (example in GVL_MSG.LOG_FILE)
  _pDirRoot     : POINTER TO STRING(255);     // see GVL_MSG.LOG_DIR

  _nMsgIndex    : REFERENCE TO UINT;          // Hypnos IS the only one in the village, if there are more you need more villages
  _nErrIndex    : REFERENCE TO UINT;          // Thanatos, Hypnos stern and more serious brother

  _dtLocalTime  : POINTER TO DT;
  _pMsgList     : POINTER TO ARRAY[1..GVL_MSG_XTS.MAX_MESSAGE] OF ST_Message; // attach your list here

	_rtrigReset   : Tc2_Standard.R_TRIG;
	_aWriteList   : ARRAY[1..GVL_MSG_XTS.MAX_MESSAGE] OF ST_Message;
	_sWriteData   : STRING(STR_LEN);
	_sNewLine     : STRING := '$N';
	_sTab         : STRING := '$T';
	_iCount, 
	_iStart, 
	_iEnd         : UINT;

	_fbCreateDir  : Tc2_System.FB_CreateDir;
	_sTmp         : STRING(256);
	_sFilename    : STRING(256);
	_sFolderDate  : STRING;
	_bFileCreated : BOOL;

	_fbFileOpen   : Tc2_System.FB_FileOpen;
	_fbFileWrite  : Tc2_System.FB_FileWrite;
	_fbFileClose  : Tc2_System.FB_FileClose;
END_VAR

METHOD Builder : BOOL // string concat for length > 255
VAR_INPUT
  pInString   : POINTER TO STRING;
  pOutString  : POINTER TO STRING(STR_LEN);
  Length      : UINT;
END_VAR
VAR
  Counter     : UDINT;
  pInWork     : POINTER TO BYTE;
  pOutWork    : POINTER TO BYTE;
END_VAR
pOutWork := pOutString;
pInWork := pInString;
Counter := 0;

(*check termination*)
WHILE (pOutWork^ <> 0) AND
      (Counter < STR_LEN+1)
DO
  Counter := Counter + 1;
  pOutWork := pOutWork + 1;
END_WHILE

(* append only if data fits into output *)
IF (Counter + Length < STR_LEN+1)
THEN

  (* append data *)
  FOR Counter := 1 TO Length
  DO
    pOutWork^ := pInWork^;
    pOutWork := pOutWork + 1;
    pInWork := pInWork + 1;
  END_FOR

  (* terminate *)
  pOutWork := pOutWork + 1;
  pOutWork^ := 0;
END_IF
END_METHOD

METHOD Check : BOOL
VAR_INPUT
END_VAR

IF NOT (_dtLocalTime <> 0)
THEN
  _eCheck       := E_MESSAGE_CHECK.POINTER_TIME_INVALID;
  RETURN;
END_IF

IF NOT (_pMsgList <> 0)
THEN
  _eCheck       := E_MESSAGE_CHECK.POINTER_LIST_INVALID;
  RETURN;
END_IF

IF NOT (_pFileRoot <> 0)
THEN
  _eCheck       := E_MESSAGE_CHECK.POINTER_ROOT_FILE_INVALID;
  RETURN;
END_IF

IF NOT (_pDirRoot <> 0)
THEN
  _eCheck       := E_MESSAGE_CHECK.POINTER_ROOT_DIR_INVALID;
  RETURN;
END_IF

IF NOT __ISVALIDREF(_nMsgIndex)
THEN
  _eCheck       := E_MESSAGE_CHECK.POINTER_MSG_IDX_INVALID;
  RETURN;
END_IF

IF NOT __ISVALIDREF(_nErrIndex)
THEN
  _eCheck       := E_MESSAGE_CHECK.POINTER_ERR_IDX_INVALID;
  RETURN;
END_IF


_eCheck         := E_MESSAGE_CHECK.CHECK_DONE;
Check           := TRUE;
END_METHOD

METHOD Device_to_String : string
VAR_INPUT
  eMsgDevice    : e_Device;
END_VAR
VAR
  sId                 : STRING := '_ID_';
  nId                 : UDINT;
END_VAR
IF (eMsgDevice < e_device.General)
THEN
  // below general case
  nId := TO_UDINT(eMsgDevice);
  //sId := concat(sId, TO_STRING(nId));

  //Device_to_String := concat(TO_STRING(eMsgDevice), sId);
  Device_to_String := TO_STRING(eMsgDevice);

ELSE
  IF (eMsgDevice >= e_Device.DataProduct)
  THEN
    nId := eMsgDevice MOD e_Device.DataProduct;
    sId := concat(sId, TO_STRING(nId));
 
    Device_to_String := concat(TO_STRING(e_Device.DataProduct), sId);

  ELSIF (eMsgDevice >= e_Device.Application)
  THEN
    nId := eMsgDevice MOD e_Device.Application;
    sId := concat(sId, TO_STRING(nId));
 
    Device_to_String := concat(TO_STRING(e_Device.Application), sId);

  ELSIF (eMsgDevice >= e_Device.TicketListCtrl)
  THEN
    nId := eMsgDevice MOD e_Device.TicketListCtrl;
    sId := concat(sId, TO_STRING(nId));
 
    Device_to_String := concat(TO_STRING(e_Device.TicketListCtrl), sId);

  ELSIF (eMsgDevice >= e_Device.ProcessListCtrl)
  THEN
    nId := eMsgDevice MOD e_Device.ProcessListCtrl;
    sId := concat(sId, TO_STRING(nId));
 
    Device_to_String := concat(TO_STRING(e_Device.ProcessListCtrl), sId);

  ELSIF (eMsgDevice >= e_Device.Process)
  THEN
    nId := eMsgDevice MOD e_Device.Process;
    sId := concat(sId, TO_STRING(nId));
 
    Device_to_String := concat(TO_STRING(e_Device.Process), sId);

  ELSIF (eMsgDevice >= e_Device.MetricsAxis)
  THEN
    nId := eMsgDevice MOD e_Device.MetricsAxis;
    sId := concat(sId, TO_STRING(nId));
 
    Device_to_String := concat(TO_STRING(e_device.MetricsAxis), sId);

  ELSIF (eMsgDevice >= e_Device.MetricsXts)
  THEN
    nId := eMsgDevice MOD e_Device.MetricsXts;
    sId := concat(sId, TO_STRING(nId));
 
    Device_to_String := concat(TO_STRING(e_device.MetricsXts), sId);

  ELSIF (eMsgDevice >= e_device.XfcAxis)
  THEN
    nId := eMsgDevice MOD e_device.XfcAxis;
    sId := concat(sId, TO_STRING(nId));
 
    Device_to_String := concat(TO_STRING(e_device.XfcAxis), sId);

  ELSIF (eMsgDevice >= e_device.Axis)
  THEN
    nId := eMsgDevice MOD e_device.Axis;
    sId := concat(sId, TO_STRING(nId));
 
    Device_to_String := concat(TO_STRING(e_device.Axis), sId);

  ELSIF (eMsgDevice >= e_device.NciChannelCtrl)
  THEN
    nId := eMsgDevice MOD e_device.NciChannelCtrl;
    sId := concat(sId, TO_STRING(nId));
 
    Device_to_String := concat(TO_STRING(e_device.NciChannelCtrl), sId);

  ELSIF (eMsgDevice >= e_device.NciChannel)
  THEN
    nId := eMsgDevice MOD e_device.NciChannel;
    sId := concat(sId, TO_STRING(nId));
 
    Device_to_String := concat(TO_STRING(e_device.NciChannel), sId);

  ELSIF (eMsgDevice >= e_Device.Camming)
  THEN
    nId := eMsgDevice MOD e_Device.Camming;
    sId := concat(sId, TO_STRING(nId));
 
    Device_to_String := concat(TO_STRING(e_device.Camming), sId);

  ELSIF (eMsgDevice >= e_Device.XtsStation)
  THEN
    nId := eMsgDevice MOD e_Device.XtsStation;
    sId := concat(sId, TO_STRING(nId));
 
    Device_to_String := concat(TO_STRING(e_device.XtsStation), sId);

  ELSIF (eMsgDevice >= e_Device.XfcTouchProbe)
  THEN
    nId := eMsgDevice MOD e_Device.XfcTouchProbe;
    sId := concat(sId, TO_STRING(nId));
 
    Device_to_String := concat(TO_STRING(e_device.XfcTouchProbe), sId);

  ELSIF (eMsgDevice >= e_Device.XfcTriggerBox)
  THEN
    nId := eMsgDevice MOD e_Device.XfcTriggerBox;
    sId := concat(sId, TO_STRING(nId));
 
    Device_to_String := concat(TO_STRING(e_device.XfcTriggerBox), sId);

  ELSIF (eMsgDevice >= e_Device.XtsTransportUnit)
  THEN
    nId := eMsgDevice MOD e_Device.XtsTransportUnit;
    sId := concat(sId, TO_STRING(nId));
 
    Device_to_String := concat(TO_STRING(e_device.XtsTransportUnit), sId);

  ELSIF (eMsgDevice >= e_Device.MoverCtrl)
  THEN
    nId := eMsgDevice MOD e_Device.MoverCtrl;
    sId := concat(sId, TO_STRING(nId));
 
    Device_to_String := concat(TO_STRING(e_device.MoverCtrl), sId);

  ELSIF (eMsgDevice >= e_Device.Mover)
  THEN
    nId := eMsgDevice MOD e_Device.Mover;
    sId := concat(sId, TO_STRING(nId));
 
    Device_to_String := concat(TO_STRING(e_device.Mover), sId);

  ELSIF (eMsgDevice >= e_Device.XpuCtrl)
  THEN
    nId := eMsgDevice MOD e_Device.XpuCtrl;
    sId := concat(sId, TO_STRING(nId));
 
    Device_to_String := concat(TO_STRING(e_device.XpuCtrl), sId);

  ELSIF (eMsgDevice >= e_Device.Xpu)
  THEN
    nId := eMsgDevice MOD e_Device.Xpu;
    sId := concat(sId, TO_STRING(nId));
 
    Device_to_String := concat(TO_STRING(e_device.Xpu), sId);

  ELSIF (eMsgDevice >= e_Device.CaGroup)
  THEN
    nId := eMsgDevice MOD e_Device.CaGroup;
    sId := concat(sId, TO_STRING(nId));
 
    Device_to_String := concat(TO_STRING(e_device.CaGroup), sId);

  ELSIF (eMsgDevice >= e_Device.General)
  THEN
    nId := eMsgDevice MOD e_Device.General;
    //sId := concat(sId, TO_STRING(nId));
 
    Device_to_String := TO_STRING(e_device.General);

  ELSE
    Device_to_String := TO_STRING(eMsgDevice);
  END_IF
END_IF
END_METHOD

PROPERTY DirRoot : POINTER to string(255)
SET
_pDirRoot := DirRoot;
END_SET
END_PROPERTY

PROPERTY ErrorIndex : reference to uint
SET
_nErrIndex  REF= ErrorIndex;
END_SET
END_PROPERTY

PROPERTY FileRoot : pointer to string(255)
SET
_pFileRoot := FileRoot;
END_SET
END_PROPERTY

METHOD FolderDate : STRING
VAR_INPUT
	LocalTime   : POINTER TO DT;
END_VAR
VAR
	sTmp        : STRING;
END_VAR
IF NOT (LocalTime <> 0)
THEN
	FolderDate := 'NULL';
	RETURN;
END_IF

sTmp := DT_TO_STRING(LocalTime^);

// cut off #dt literal
sTmp := right(sTmp, len(sTmp)-3);

sTmp := replace(sTmp, '_', 1, 5);
sTmp := replace(sTmp, '_', 1, 8);

sTmp := left(sTmp,10);	// year_month_day

FolderDate := sTmp;
END_METHOD

PROPERTY LocalTime : pointer to DT
SET
_dtLocalTime := LocalTime;
END_SET
END_PROPERTY

PROPERTY MessageIndex : reference to uint
SET
_nMsgIndex   REF= MessageIndex;
END_SET
END_PROPERTY

PROPERTY MsgList : pointer to ARRAY[1..GVL_MSG_XTS.MAX_MESSAGE] OF st_message
SET
_pMsgList := MsgList;
END_SET
END_PROPERTY

METHOD StringLen : UINT // 	string length for len > 255
VAR_INPUT
  pInString		: POINTER TO STRING(STR_LEN);
END_VAR
VAR
	Counter			: UINT;
	pInWork			: POINTER TO BYTE;
END_VAR
pInWork := pInString;
Counter := 0;

WHILE (pInWork^ <> 0) AND
			(Counter < STR_LEN)
DO
	Counter := Counter + 1;
	pInWork := pInWork + 1;
END_WHILE

StringLen := Counter;
END_METHOD

METHOD WriteData  : e_progress
VAR_INPUT
  bExecute        : BOOL;
END_VAR
VAR_INST
  _eState         : e_progress;
  _bError         : BOOL;
  _nErrorId       : UDINT;
END_VAR
IF NOT bExecute
THEN
  _eState                     := E_PROGRESS.PROGRESS_INIT;
END_IF

CASE _eState 
OF

	E_PROGRESS.PROGRESS_INIT:
    _fbFileOpen(
        sPathName             := _sFilename, 
        nMode                 := FOPEN_MODEAPPEND OR FOPEN_MODEPLUS, 
        ePath                 := PATH_GENERIC, 
        bExecute              := FALSE, 
        tTimeout              := T#5S);

    _fbFileWrite(
        hFile                 := _fbFileOpen.hFile, 
        pWriteBuff            := ADR(_sWriteData), 
        cbWriteLen            := StringLen(ADR(_sWriteData)),
        bExecute              := FALSE, 
        tTimeout              := T#5S);

    _fbFileClose(
        hFile                 := _fbFileOpen.hFile, 
        bExecute              := FALSE, 
        tTimeout              := T#5S);


		IF bExecute
		THEN
      _nErrorId               := 0;
      _eState                 := E_PROGRESS.PROGRESS_BUSY;
		END_IF

	E_PROGRESS.PROGRESS_BUSY:
		_fbFileOpen(bExecute      := TRUE);

    IF _fbFileOpen.bError
    THEN
      _nErrorId               := _fbFileOpen.nErrId;
      _eState                 := E_PROGRESS.PROGRESS_ERROR;

		ELSIF _fbFileOpen.bBusy
		THEN
      _eState                 := E_PROGRESS.PROGRESS_PREPARE;
		END_IF

	E_PROGRESS.PROGRESS_PREPARE:
		_fbFileOpen(bExecute      := TRUE);
		IF NOT _fbFileOpen.bBusy
		THEN
		  _fbFileOpen(bExecute    := FALSE);
      _eState                 := E_PROGRESS.PROGRESS_STARTUP;
		END_IF

	E_PROGRESS.PROGRESS_STARTUP:
    _fbFileWrite(
        hFile                 := _fbFileOpen.hFile, 
        pWriteBuff            := ADR(_sWriteData), 
        cbWriteLen            := StringLen(ADR(_sWriteData)),
        bExecute              := TRUE, 
        tTimeout              := T#5S);

    IF _fbFileWrite.bError
    THEN
      _nErrorId               := _fbFileWrite.nErrId;
      _eState                 := E_PROGRESS.PROGRESS_ERROR;

		ELSIF _fbFileWrite.bBusy
		THEN
      _eState                 := E_PROGRESS.PROGRESS_CHECK;
		END_IF

	E_PROGRESS.PROGRESS_CHECK:
	  _fbFileWrite(bExecute     := TRUE);
		IF NOT _fbFileWrite.bBusy
		THEN
			_fbFileWrite(bExecute   := FALSE);
      _eState                 := E_PROGRESS.PROGRESS_OCCUPIED;
		END_IF

	E_PROGRESS.PROGRESS_OCCUPIED:
    _fbFileClose(
        hFile                 := _fbFileOpen.hFile, 
        bExecute              := TRUE, 
        tTimeout              := T#5S);

    IF _fbFileClose.bError
    THEN
      _nErrorId               := _fbFileClose.nErrId;
      _eState                 := E_PROGRESS.PROGRESS_ERROR;

		ELSIF _fbFileClose.bBusy
		THEN
      _eState                 := E_PROGRESS.PROGRESS_WORKING;
		END_IF

	E_PROGRESS.PROGRESS_WORKING:
    _fbFileClose(bExecute     := TRUE);
		IF NOT _fbFileClose.bBusy
		THEN
			_fbFileClose(bExecute   := FALSE);
      _eState                 := E_PROGRESS.PROGRESS_DONE;
		END_IF

END_CASE
CASE _eState
OF
  E_PROGRESS.PROGRESS_ERROR:
		_fbFileOpen (bExecute     := FALSE);
    _fbFileWrite(bExecute     := FALSE);
    _fbFileClose(bExecute     := FALSE);


END_CASE




WriteData                     := _eState;
END_METHOD

END_FUNCTION_BLOCK

// ---- _MSG/class/fb_LocalTime.TcPOU
//-----------------------------------------------------------------------------------------------
//
//  As time goes by...
//
//  HAUD 2026 07 23
//  - timezone to match UTC device time.
//-----------------------------------------------------------------------------------------------
FUNCTION_BLOCK fb_LocalTime
VAR
  _eState                 : e_progress;   // self startup state, reaches WORKING when done.
  _stSystemtime           : Tc2_Utilities.TIMESTRUCT;

  _stUtcTime              : Tc2_Utilities.T_FILETIME64; // CPU time as 64bit ULINT, meant to be used for measurement
  _sUtcTime               : STRING;
  _dtUtcTime              : DT;

  _stLocalTime            : Tc2_Utilities.T_FILETIME64; // In every wood, in every spring,there is a different green.
  _sLocalTime             : STRING;
  _dtLocalTime            : DT;

  _eTimeZoneId            : Tc2_Utilities.E_TimeZoneID;
  _stTimeZoneInfo         : Tc2_Utilities.ST_TimeZoneInformation;
  _fbGetTimeZoneInfo      : Tc2_Utilities.FB_GetTimeZoneInformation;
  _fbFileTimeToLocalTime  : Tc2_Utilities.FB_FileTime64ToTzSpecificLocalTime;
  _nErrorId               : UDINT;
  _bError                 : BOOL;
END_VAR

//-----------------------------------------------------------------------------------------------
// infosys: https://infosys.beckhoff.com/english.php?content=../content/1033/tcplclib_tc2_system/3622991755.html&id=6591934602709167291
//-----------------------------------------------------------------------------------------------
// This function can be used to read the operating system timestamp. 
// The timestamp is a 64-bit integer value, with an accuracy of 100 ns, 
// which is updated with every call of the PLC. 
// Among other things, it can be used for timing tasks or time measurements. 
// One unit corresponds to 100 ns. 
// The time represents the number of 100 ns intervals since January 1, 1601 (UTC).
//-----------------------------------------------------------------------------------------------
//-----------------------------------------------------------------------------------------------
_stUtcTime                      := F_GetSystemTime(); // UTC time, no delay --> CPU time direct
//-----------------------------------------------------------------------------------------------
//-----------------------------------------------------------------------------------------------
// build UTC time
_sUtcTime                       := SYSTEMTIME_TO_STRING( FILETIME64_TO_SYSTEMTIME( _stUtcTime ));
_dtUtcTime                      := systemtime_to_dt    ( FILETIME64_TO_SYSTEMTIME( _stUtcTime ));
//-----------------------------------------------------------------------------------------------
//-----------------------------------------------------------------------------------------------
// state machine for getting timezone information and add the offset to UTC time
//-----------------------------------------------------------------------------------------------
CASE _eState
OF
  E_PROGRESS.PROGRESS_INVALID:
    _eState                     := E_PROGRESS.PROGRESS_INIT;
    _fbGetTimeZoneInfo(
                      sNetID    := '', 
                      bExecute  := FALSE,
                      bError    => _bError,
                      nErrID    => _nErrorId, 
                      tzID      => _eTimeZoneId, 
                      tzInfo    => _stTimeZoneInfo);
END_CASE
//---------------------------------------------------------------------------------------------
//---------------------------------------------------------------------------------------------
CASE _eState
OF
  E_PROGRESS.PROGRESS_INIT:
    _fbGetTimeZoneInfo(
                      sNetID    := '', 
                      bExecute  := TRUE,
                      bError    => _bError,
                      nErrID    => _nErrorId, 
                      tzID      => _eTimeZoneId, 
                      tzInfo    => _stTimeZoneInfo);

    IF (_fbGetTimeZoneInfo.bBusy)
    THEN
      _eState                   := E_PROGRESS.PROGRESS_PREPARE;
    END_IF
END_CASE
//---------------------------------------------------------------------------------------------
//---------------------------------------------------------------------------------------------
CASE _eState
OF
  E_PROGRESS.PROGRESS_PREPARE:
    _fbGetTimeZoneInfo(
                      sNetID    := '', 
                      bExecute  := TRUE,
                      bError    => _bError,
                      nErrID    => _nErrorId, 
                      tzID      => _eTimeZoneId, 
                      tzInfo    => _stTimeZoneInfo);

    IF NOT (_fbGetTimeZoneInfo.bBusy)
    THEN
      _fbGetTimeZoneInfo(
                      sNetID    := '', 
                      bExecute  := FALSE);

      _eState                   := E_PROGRESS.PROGRESS_WORKING;
    END_IF
END_CASE
//---------------------------------------------------------------------------------------------
//---------------------------------------------------------------------------------------------
CASE _eState
OF
  E_PROGRESS.PROGRESS_WORKING:
    _fbFileTimeToLocalTime(
                      in        := _stUtcTime, 
                      tzInfo    := _stTimeZoneInfo, 
                      out       => _stLocalTime, 
                      eTzID     => _eTimeZoneId);

  // build local time
  _stSystemtime                 := FILETIME64_TO_SYSTEMTIME( _stLocalTime );
  _sLocalTime                   := SYSTEMTIME_TO_STRING    ( _stSystemtime );
  _dtLocalTime                  := systemtime_to_dt        ( _stSystemtime );


  IF (_stSystemtime.wHour   = 0) AND
     (_stSystemtime.wMinute = 0) AND
     (_stSystemtime.wSecond = 0)
  THEN
    //  The passing seasons are but ripples ever repeated in the long long stream.
    _eState                     := E_PROGRESS.PROGRESS_INIT;
  END_IF
END_CASE
//---------------------------------------------------------------------------------------------
//---------------------------------------------------------------------------------------------

METHOD FolderDate : STRING
VAR_INPUT
	LocalTime   : POINTER TO DT;
END_VAR
VAR
	sTmp        : STRING;
END_VAR
IF NOT (LocalTime <> 0)
THEN
	FolderDate := 'NULL';
	RETURN;
END_IF

sTmp := DT_TO_STRING(LocalTime^);

// cut off #dt literal
sTmp := right(sTmp, len(sTmp)-3);

sTmp := replace(sTmp, '_', 1, 5);
sTmp := replace(sTmp, '_', 1, 8);

sTmp := left(sTmp,10);	// year_month_day

FolderDate := sTmp;
END_METHOD

PROPERTY LocalTime : DT
GET
LocalTime := _dtLocalTime;
END_GET
END_PROPERTY

PROPERTY LocalTimeString : string
GET
IF (len(_sLocalTime) >1)
THEN
  LocalTimeString := _sLocalTime;
ELSE
  LocalTimeString := _sUtcTime;
END_IF
END_GET
END_PROPERTY

PROPERTY State : e_progress
GET
State := _eState;
END_GET
END_PROPERTY

PROPERTY UtcTime : DT
GET
UtcTime := _dtUtcTime;
END_GET
END_PROPERTY

PROPERTY UtcTimeString : string
GET
UtcTimeString := _sUtcTime;
END_GET
END_PROPERTY

END_FUNCTION_BLOCK

// ---- APPLICATION/MAIN_APP.TcPOU
//---------------------------------------------------------------------------------------------------------------
//
//  HAUD 2024.04.26
//
//  - APPLICATION
//    - explicit simple example PRG for setting up application
//      - no additional interfaces or encapsulations
//      - works dirEctly on GVL_XTS namespace Ctrl/State structs
//      - no error handling, reset application from start
//
//  - Application controls:
//    - XtsTransport
//      - GVL_XTS.TransportCtrl
//      - GVL_XTS.TransportState
//
//    - Xts Stations
//      - GVL_XTS.StationCtrl[]
//      - GVL_XTS.StationState[]
//      - see MAIN.StationParameterInit for XtsStation parameters.
//        - Intention: for developing a transport layer, 
//                      the station parameters are part of the XTS, 
//                      the application primarily handles handshakes with XtsStations
//
//  - Application
//    - 5 single XtsStations
//      - automated handshakes 
//      - process with TON
//      - static targets
//
//---------------------------------------------------------------------------------------------------------------
// This SOFTWARE is provided as an Example by THE PROVIDER "as is" and "with all faults." THE PROVIDER makes no 
// representations or warranties of any kind concerning the safety, suitability, lack of viruses, inaccuracies, 
// typographical errors, or other harmful components of this SOFTWARE. There are inherent dangers in the use of 
// any software, and you are solely responsible for determining whether this SOFTWARE is compatible with your 
// equipment and other software installed on your equipment. You are also solely responsible for the protection 
// of your equipment and backup of your data, and THE PROVIDER will not be liable for any damages you may suffer 
// in connection with using, modifying, or distributing this SOFTWARE.
//---------------------------------------------------------------------------------------------------------------
PROGRAM MAIN_APP
VAR
  eInitXts  AT %I*    : E_PROGRESS;
  eInit               : E_PROGRESS;
  bStart              : BOOL;   // XtsTransport is initialized, CAGroup is built, All movers are enabled, XtsStations are cleared, XtsTransport base position for all movers is commanded, XtsStations are handshaked with timer
  bReset              : BOOL;   // All Xts Stations are cleared, requires new start

  nState              : UINT;   // state var for application

  tonProcess          : ARRAY[1..MAX_STATION] OF Tc2_Standard.TON;
  tProcess            : ARRAY[1..MAX_STATION] OF TIME;

  // work vars
  nStation            : UINT;
  nTarget             : ARRAY[1..MAX_STATION] OF UINT;  // contains target the station is sending the mover to, after process handshake was done

  JobResult           : E_PROGRESS;

  // example work vars
  eTransportState,
  eTransportStateOld  : E_XTS_TRANSPORT_STATE;

  eExecState          : E_XTS_TRANSPORT_STATE;
  eExecResult         : e_progress;
  stMsg               : ST_Message;
END_VAR

//-----------------------------------------------------------------------------
// wait for initialization to be complete before work may start
//-----------------------------------------------------------------------------
IF NOT (eInitXts = E_PROGRESS.PROGRESS_DONE)
THEN
  eInit                               := E_PROGRESS.PROGRESS_INIT;
  bReset                              := FALSE;
  bStart                              := FALSE;
  nState                              := 0;
  RETURN;
END_IF
//-----------------------------------------------------------------------------
// fetch reset anytime
//-----------------------------------------------------------------------------
IF bReset
THEN
  bReset                              := FALSE;
  bStart                              := FALSE;
  nState                              := 9000;  // states for clearing XtsTransport
END_IF
//-----------------------------------------------------------------------------
// basic example procedures to startup the XTS_TRANSPORT_LAYER
//  - this is only for showing thw basic handshake mechanics 
//  - this not a production ready state machine 
//-----------------------------------------------------------------------------
CASE nState 
OF
  0:                                  // first PLC cycle
    eInit                             := E_PROGRESS.PROGRESS_INIT;
    nState                            := 1;
    FOR nStation := 1 TO MAX_STATION
    DO
      tProcess[nStation]              := T#650MS;
      nTarget [nStation]              := SEL(nStation<MAX_STATION, 1, nStation+1);
    END_FOR

  1:
    // do other init stuff here
    eInit                             := E_PROGRESS.PROGRESS_DONE;
    nState                            := 10;

  10:                                 // starts from here
    IF bStart
    THEN
      nState                          := 100; // let's go
    END_IF
    
  100:                                // clear interface
    GVL_XTS.XtsTransportCtrl.Cmd      := E_XTS_TRANSPORT_CTRL.CMD_NULL;
    nState                            := 110;

  110:                                // check initialization of XtsTransport, wait for either MoverDetection being valid or OperationMode.Simulation
    IF (GVL_XTS.XtsTransportState.XpuInfo.IdDetectionValid) OR
       (GVL_XTS.XtsTransportState.XpuInfo.OperationMode = OperationMode.Simulation)
    THEN
      // now XtsTransport is initialized, cyclic plausibility checks on Xpu are active
      nState                          := 120;
    END_IF

  120:                                // clear group for defined start situation
    GVL_XTS.XtsTransportCtrl.Cmd      := E_XTS_TRANSPORT_CTRL.CMD_GROUP_CLEAR;

    IF (GVL_XTS.XtsTransportState.State = E_XTS_TRANSPORT_STATE.TRANSPORT_GROUP_CLEAR + E_PROGRESS.PROGRESS_ERROR)
    THEN
      nState                          := 9033;

    ELSIF (GVL_XTS.XtsTransportState.State = E_XTS_TRANSPORT_STATE.TRANSPORT_GROUP_CLEAR + E_PROGRESS.PROGRESS_DONE)
    THEN
      // CA Group is now in defined error free state
      nState                          := 130;
    END_IF

  130:                                // build Collision Avoidance group with all movers
    GVL_XTS.XtsTransportCtrl.Cmd      := E_XTS_TRANSPORT_CTRL.CMD_GROUP_BUILD;

    IF (GVL_XTS.XtsTransportState.State = E_XTS_TRANSPORT_STATE.TRANSPORT_GROUP_BUILD + E_PROGRESS.PROGRESS_ERROR)
    THEN
      nState                          := 9044;

    ELSIF (GVL_XTS.XtsTransportState.State = E_XTS_TRANSPORT_STATE.TRANSPORT_GROUP_BUILD + E_PROGRESS.PROGRESS_DONE)
    THEN
      // CA Group contains all movers now
      // GVL_XTS.XtsTransportState.GroupInfo.AxisCount = MAX_MOVER
      nState                          := 140;
    END_IF

  140:                                // enable CA Group
    GVL_XTS.XtsTransportCtrl.Cmd      := E_XTS_TRANSPORT_CTRL.CMD_GROUP_ENABLE;

    IF (GVL_XTS.XtsTransportState.State = E_XTS_TRANSPORT_STATE.TRANSPORT_GROUP_ENABLE + E_PROGRESS.PROGRESS_ERROR)
    THEN
      nState                          := 9011;

    ELSIF (GVL_XTS.XtsTransportState.State = E_XTS_TRANSPORT_STATE.TRANSPORT_GROUP_ENABLE + E_PROGRESS.PROGRESS_DONE)
    THEN
      // GVL_XTS.XtsTransportState.GroupInfo.CaGroupState = mcGroupStateNotReady
      nState                          := 150;
    END_IF

  150:                                // enable all movers
    GVL_XTS.XtsTransportCtrl.Cmd      := E_XTS_TRANSPORT_CTRL.CMD_MOVER_ENABLE;

    IF (GVL_XTS.XtsTransportState.State = E_XTS_TRANSPORT_STATE.TRANSPORT_MOVER_ENABLE + E_PROGRESS.PROGRESS_ERROR)
    THEN
      nState                          := 9011;

    ELSIF (GVL_XTS.XtsTransportState.State = E_XTS_TRANSPORT_STATE.TRANSPORT_MOVER_ENABLE + E_PROGRESS.PROGRESS_DONE)
    THEN
      // GVL_XTS.XtsTransportState.GroupInfo.CaGroupState = mcGroupStateStandby
      nState                          := 160;
    END_IF

  160:                                // command all movers to startup position
    GVL_XTS.XtsTransportCtrl.Cmd      := E_XTS_TRANSPORT_CTRL.CMD_TRANSPORT_START;

    IF (GVL_XTS.XtsTransportState.State = E_XTS_TRANSPORT_STATE.TRANSPORT_START + E_PROGRESS.PROGRESS_DONE)
    THEN
      // all XtsStations are cleared
      // all movers are now waiting at GVL_XTS.XtsTransport.StartStationIndex
      // all movers are entered into GVL_XTS.StationList[GVL_XTS.XtsTransport.StartStationIndex]._stList 
      nState                          := 170;
    END_IF

  170:
    nState                            := 1000;

  1000:                               // automatic handshakes with XtsStations
    FOR nStation := 1 TO MAX_STATION
    DO
      CASE GVL_XTS.StationState[nStation].State
      OF
        //-------------------------------------------------------------------------------------
        E_STATION_STATE.STATION_DISABLE:          // switch on XtsStation
          GVL_XTS.StationCtrl[nStation].Cmd     := E_STATION_CTRL.STATION_ENABLE;

        //-------------------------------------------------------------------------------------
        E_STATION_STATE.STATION_MOVER_ENTER:      // let mover enter
          // mover was detected in list and station is asking for mover entry
          IF (tProcess[nStation] < T#10MS)
          THEN
            // this is an example! make the decision whether to work or not in your world, then fire the command you have chosen.
            GVL_XTS.StationCtrl[nStation].Cmd   := E_STATION_CTRL.STATION_MOVER_SEND;     // no process handshake, direct state change to MOVER_OUT
          ELSE 
            GVL_XTS.StationCtrl[nStation].Cmd   := E_STATION_CTRL.STATION_MOVER_ENTER;    // allow entry
          END_IF

        //-------------------------------------------------------------------------------------
        E_STATION_STATE.STATION_PROCESS_START:    // first process handshake, clear timer
          // mover has arrived and is in standstill, ready for process 
          tonProcess[nStation](
                              IN                :=FALSE, 
                              PT                :=tProcess[nStation]);
          GVL_XTS.StationCtrl[nStation].Cmd     := E_STATION_CTRL.STATION_PROCESS_START;  // regular 'double' handshake for you to organise your process procedure

//          GVL_XTS.StationCtrl[nStation].Cmd     := E_STATION_CTRL.STATION_PROCESS_DONE;   // regular 'single' handshake for you to organise your process procedure
//          GVL_XTS.StationCtrl[nStation].Cmd     := E_STATION_CTRL.STATION_MOVER_OUT;      // the shortest straw has been pulled for you - if you trigger this you MUST be sure that your target data is valid


        //-------------------------------------------------------------------------------------
        E_STATION_STATE.STATION_PROCESS_DONE:     // second process handshake, timer runs now
          tonProcess[nStation](
                              IN                :=TRUE, 
                              PT                :=tProcess[nStation]);
          IF tonProcess[nStation].Q
          THEN
            GVL_XTS.StationCtrl[nStation].nTargetStation  := TO_USINT(nTarget[nStation]); // static in this example
            GVL_XTS.StationCtrl[nStation].nMask := 2#1; // bitmask for mover ticket to next XtsStation; if you use more than one StopPos[] in XtsStation

//            GVL_XTS.StationCtrl[nStation].Cmd    := E_STATION_CTRL.STATION_PROCESS_DONE; // regulear 'double' handshake

            GVL_XTS.StationCtrl[nStation].Cmd   := E_STATION_CTRL.STATION_MOVER_OUT;     // the shortest straw has been pulled for you - if you trigger this you MUST be sure that your target data is valid
          END_IF

        //-------------------------------------------------------------------------------------
        E_STATION_STATE.STATION_MOVER_OUT:        // station wants to send out mover
          // when sending out mover, the data on Ctrl struct is absolute important
          // before allowing the outfeed of the mover, the data on Ctrl struct must be entered correctly
          // Ctrl.nTargetStation allows for flexible mover transport, this is fully depending on you to make sense aside this example

          GVL_XTS.StationCtrl[nStation].nTargetStation  := TO_USINT(nTarget[nStation]); // static in this example
          GVL_XTS.StationCtrl[nStation].nMask   := 2#1; // bitmask for mover ticket to next XtsStation; if you use more than one StopPos[] in XtsStation

          GVL_XTS.StationCtrl[nStation].Cmd     := E_STATION_CTRL.STATION_MOVER_OUT;  // allow outfeed of mover

        //-------------------------------------------------------------------------------------
        E_STATION_STATE.STATION_MOVER_GONE:       // mover has travelled ReleaseDistance, XtsStation is now empty and ready for the next mover in queue
          GVL_XTS.StationCtrl[nStation].nTargetStation  := 0;                           // clear target after mover left the station
          GVL_XTS.StationCtrl[nStation].Cmd     := E_STATION_CTRL.STATION_MOVER_GONE; // last handshake for empty station
      END_CASE
    END_FOR


  9000:                               // example procedure for halting transport and clearing stations
    GVL_XTS.XtsTransportCtrl.Cmd      := E_XTS_TRANSPORT_CTRL.CMD_NULL;
    nState                            := 9010;

  9010:                               // halt all movers and clear group
    GVL_XTS.XtsTransportCtrl.Cmd      := E_XTS_TRANSPORT_CTRL.CMD_GROUP_CLEAR;

    IF (GVL_XTS.XtsTransportState.State = E_XTS_TRANSPORT_STATE.TRANSPORT_GROUP_CLEAR + E_PROGRESS.PROGRESS_ERROR)
    THEN
      nState                          := 9000;

    ELSIF (GVL_XTS.XtsTransportState.State = E_XTS_TRANSPORT_STATE.TRANSPORT_GROUP_CLEAR + E_PROGRESS.PROGRESS_DONE)
    THEN
      // CA group cleared and mover in standstill
      nState                          := 9100;
    END_IF

  9100:                               // switch off movers
    GVL_XTS.XtsTransportCtrl.Cmd      := E_XTS_TRANSPORT_CTRL.CMD_MOVER_DISABLE;

    IF (GVL_XTS.XtsTransportState.State >= E_XTS_TRANSPORT_STATE.TRANSPORT_MOVER_DISABLE + E_PROGRESS.PROGRESS_ERROR)
    THEN
      nState                          := 9200;
    END_IF

  9200:                               // clear All XtsStations
    nState                            := 9300;
    FOR nStation := 1 TO MAX_STATION
    DO
       GVL_XTS.StationCtrl[nStation].Cmd      := E_STATION_CTRL.STATION_INIT;
    END_FOR

  9300:                               // disable All XtsStations
    nState                            := 9400;   // go back to start
    FOR nStation := 1 TO MAX_STATION
    DO
       GVL_XTS.StationCtrl[nStation].Cmd      := E_STATION_CTRL.STATION_DISABLE;
    END_FOR

  9400:
    nState                            := 10;
END_CASE

END_PROGRAM

// ---- _types/f_GetState.TcPOU
// global function to extract state identifier from combined value
FUNCTION f_GetState : uint
VAR_INPUT
  state     : UINT; // combined value of identifier + e_progress
END_VAR
VAR
  _stx      : uint;
END_VAR

_stx          := state MOD E_PROGRESS.PROGRESS_INIT;

IF (_stx = 0)
THEN
  f_GetState  := state;
ELSE
  f_GetState  := _stx;
END_IF

END_FUNCTION

// ---- GlobalTextList.TcGTLO
TEXTLIST GlobalTextList
  230 = ' %d'
  30 = ' Act Pos Absolute'
  518 = ' Act Pos Modulo'
  493 = ' Avoiding Collision'
  587 = ' Coupled'
  690 = ' Enabled'
  968 = ' Error'
  144 = ' MOVER command'
  271 = ' MOVER result:  %s'
  268 = ' MOVER state:   %s'
  484 = ' nError ID'
  912 = ' Set Acceleration'
  819 = ' Set Delta'
  464 = ' Set Distance'
  1025 = ' Set Gap'
  363 = ' Set Jerk'
  376 = ' Set Override'
  1069 = ' Set Position'
  859 = ' Set Velocity'
  123 = ' Standstill'
  17 = ' STATION_ENABLE'
  34 = ' STATION_MOVER_ENTER'
  452 = ' STATION_MOVER_GONE'
  75 = ' STATION_MOVER_OUT'
  598 = ' STATION_PROCESS_DONE'
  750 = ' STATION_PROCESS_START'
  727 = ' Target Pos Absolute'
  397 = ' Target Pos Modulo'
  294 = '%.2f'
  191 = '%d'
  836 = '%s'
  704 = 'All Positions Valid'
  562 = 'AllAxisStanding'
  878 = 'AxisCount Enabled: %d'
  162 = 'AxisCount: %d'
  516 = 'CA GroupInfo'
  929 = 'Control'
  707 = 'CyclicCheck: %s'
  660 = 'DC Link All Modules'
  843 = 'Detected AxisCount: %d'
  772 = 'Expected AxisCount: %d'
  48 = 'GroupDisabled'
  915 = 'GroupError'
  495 = 'GroupErrorId: %d'
  975 = 'GroupErrorStop'
  300 = 'GroupMoving'
  807 = 'GroupNotReady'
  438 = 'GroupStandby'
  226 = 'GroupStatusBusy'
  204 = 'GroupStatusValid'
  973 = 'GroupStopping'
  680 = 'ID Detection Active'
  238 = 'ID Detection Error'
  526 = 'ID Detection Mode: %s'
  29 = 'ID Detection Valid'
  211 = 'Info Act Pos Absolute'
  586 = 'Info Act Pos Modulo'
  21 = 'Info Mover Avoiding Collision'
  282 = 'Info Mover Coupled'
  398 = 'Info Mover Enabled'
  751 = 'Info Mover Error'
  907 = 'Info Mover Standstill'
  480 = 'Info nError ID'
  922 = 'Info Target Pos Absolute'
  16 = 'Info Target Pos Modulo'
  779 = 'Mask: %s'
  726 = 'McGroupState:      %s'
  974 = 'MOVER command'
  387 = 'Mover ID: %d'
  297 = 'Mover Position Assignement: %s'
  840 = 'MOVER result:  %s'
  53 = 'MOVER state:   %s'
  145 = 'nMover: %d'
  756 = 'nMoverSelected: %d'
  427 = 'Offset: %.3f'
  312 = 'Operation Mode: %s'
  320 = 'Queue: %d'
  91 = 'Set Acceleration'
  399 = 'Set Delta'
  382 = 'Set Distance'
  757 = 'Set Gap'
  934 = 'Set Jerk'
  201 = 'Set Override'
  936 = 'Set Position'
  62 = 'Set Velocity'
  231 = 'State'
  567 = 'Target Station: %d'
  227 = 'XpuResult:   %s'
  96 = 'XpuState:    %s'
  884 = 'XTS Station'
  572 = 'XTS Transport Check:  %s'
  500 = 'XTS Transport Command'
  395 = 'XTS Transport Result: %s'
  798 = 'XTS Transport State:  %s'
END_TEXTLIST

